// TIA Portal V16 export
// export: Created 2021-11-12T13:32:01.6049772Z, ExportSetting WithDefaults, DisplayName Totally Integrated Automation Portal, DisplayVersion V16 Update 3, DisplayName TIA Portal Version Control Interface, DisplayVersion V16 Update 2, DisplayName TIA Portal Openness, DisplayVersion V16 Update 3, DisplayName SINAMICS Startdrive Advanced, DisplayVersion V16 Update 5, DisplayName SINAMICS Startdrive G130, G150, S120, S150, SINAMICS MV, S210, DisplayVersion V16 Update 5, DisplayName SINAMICS Startdrive G110M, G120, G120C, G120D, G120P, G115D, DisplayVersion V16 Update 5, DisplayName STEP 7 Professional, DisplayVersion V16 Update 3, DisplayName STEP 7 Safety, DisplayVersion V16, DisplayName WinCC UA Professional, DisplayVersion V16 Update 3
FUNCTION_BLOCK "Station 110"   // FB53, LAD
{ S7_Optimized_Access := 'TRUE' }
VERSION : 0.1
// stored: AutoNumber true, IsIECCheckEnabled false, IsRetainMemResEnabled false, MemoryReserve 100, SetENOAutomatically false, UDAEnableTagReadback false
   VAR
      SF_Alarm1 : "STD_DI_Mon";
      SF_Alarm2 { S7_SetPoint := 'True'} : "STD_DI_Mon";
      SF_Alarm3 { S7_SetPoint := 'True'} : "STD_DI_Mon";
      SF_Alarm4 { S7_SetPoint := 'True'} : "STD_DI_Mon";
      SF_Alarm5 { S7_SetPoint := 'True'} : "STD_DI_Mon";
      SF_Alarm6 { S7_SetPoint := 'True'} : "STD_DI_Mon";
      SF_Alarm7 { S7_SetPoint := 'True'} : "STD_DI_Mon";
      SF_Alarm8 { S7_SetPoint := 'True'} : "STD_DI_Mon";
      SF_Alarm9 { S7_SetPoint := 'True'} : "STD_DI_Mon";
      SF_Alarm10 { S7_SetPoint := 'True'} : "STD_DI_Mon";
      SF_Alarm11 { S7_SetPoint := 'True'} : "STD_DI_Mon";
      SF_Alarm12 { S7_SetPoint := 'True'} : "STD_DI_Mon";
      SF_Alarm13 { S7_SetPoint := 'True'} : "STD_DI_Mon";
      SF_Alarm14 { S7_SetPoint := 'True'} : "STD_DI_Mon";
      SF_Alarm15 { S7_SetPoint := 'True'} : "STD_DI_Mon";
      SF_Alarm16 { S7_SetPoint := 'True'} : "STD_DI_Mon";
      SF_Alarm17 { S7_SetPoint := 'True'} : "STD_DI_Mon";
      SF_Alarm18 { S7_SetPoint := 'True'} : "STD_DI_Mon";
      SF_Alarm19 { S7_SetPoint := 'True'} : "STD_DI_Mon";
      SF_Alarm20 { S7_SetPoint := 'True'} : "STD_DI_Mon";
      SF_Alarm21 { S7_SetPoint := 'True'} : "STD_DI_Mon";
      SF_GL01MA02 { S7_SetPoint := 'True'} : "STD_Drive1";
      SF_UH31TA01 { S7_SetPoint := 'True'} : "STD_SERVO_FESTO_CMMT";   // Aligner - frequency convertor
      SF_UC12TA01 { S7_SetPoint := 'True'} : "STD_Siemens_G120_CU240E_2_PN";
      SF_GL01BG05 { S7_SetPoint := 'True'} : "STD_Siemens_MC_Encoder";
      SF_GL01MM01 { S7_SetPoint := 'True'} : "STD_Valve2WB";
      SF_GM01MM01 { S7_SetPoint := 'True'} : "STD_Valve2WB";
      SF_GM01MM02 { S7_SetPoint := 'True'} : "STD_Valve2WB";
      SF_GM01MM03 { S7_SetPoint := 'True'} : "STD_Valve2WB";
      SF_GM01MM04 { S7_SetPoint := 'True'} : "STD_Valve2WB";
      SS_Edge : Array[0..9] of Bool;
      SF_TON_MeasDelay { S7_SetPoint := 'True'} : TON_TIME;
      SR_ConvActPos : Real;   // Conveyor - Absolute position [mm]
   END_VAR
   VAR RETAIN
      SR_ConvStopPos : Real;   // Conveyor - Demanded position [mm]
      SB1ConvInPos { ExternalAccessible := 'False'; ExternalVisible := 'False'; ExternalWritable := 'False'} : Bool := true;   // Conveyor reached position
      SB1ConvStep : Bool;   // Step is active
      SI_SeqStepNr : UInt;   // Number of active step
      SR_UH31TA01SetPos { ExternalAccessible := 'False'; ExternalVisible := 'False'; ExternalWritable := 'False'} : Real := 550.0;   // Setpoint position [mm]
   END_VAR
   VAR
      SR_MeasuredPartLenght : Real;   // Lenght of measured part [mm]
      SI_PartType : Int;   // Part type of material
      SDIPartID : DInt;   // Part Id of material
   END_VAR
   VAR_TEMP
      TS_GL01MM01 : "UDT_DriveControl";   // Stopper - valve
      TS_GL01MA01 : "UDT_DriveControl";   // Aligner - drive
      TS_GL01MA02 : "UDT_DriveControl";   // Conveyor - drive
      TS_GM01MM01 : "UDT_DriveControl";   // Lift 1 - valve
      TS_GM01MM02 : "UDT_DriveControl";   // Lift 2 - valve
      TS_GM01MM03 : "UDT_DriveControl";   // Lift 3 - valve
      TS_GM01MM04 : "UDT_DriveControl";   // Lift 4 - valve
      TS_UC12TA01 : Struct   // Conveyor
         ReqDir1 : Bool;   // Move in direction 1
         ReqDir2 : Bool;   // Move in direction 2
         AckErr : Bool;   // Acknowledge error
         SpeedSP : Real;   // Speed setpoint
      END_STRUCT;
      TS_UH31TA01 : Struct   // Aligner
         SPPos : Int;   // Aligner - setpoint
         Mode : Int;   // Aligner - mode
         HomePos : Bool;   // Aligner - home position
         WorkPos : Bool;   // Aligner - work position
      END_STRUCT;
      TR_ConvSlowPos : Real;   // Slowing position [mm]
      "TR_ConvStepTol+" : Real;   // Upper tolerance for conveyor step [mm]
      "TR_ConvStepTol-" : Real;   // Lower tolerance for conveyor step [mm]
      "TR_UH31TA01HomeTol+" : Real;   // Upper tolerance for home position [mm]
      "TR_UH31TA01HomeTol-" : Real;   // Lower tolerance for home position [mm]
      "TR_UH31TA01WorkTol+" : Real;   // Upper tolerance for work position [mm]
      "TR_UH31TA01WorkTol-" : Real;   // Lower tolerance for work position [mm]
      TR_UH31TA01ActualPos : Real;   // Absolute position [mm]
      TR_UH31TA01HomePos : Real;   // Home position [mm]
      TR_UH31TA01WorkPos : Real;   // Working position [mm]
      TR_UH31TA01SetPos : Real;   // Setpoint position [um]
      TB1PwrOk : Bool;
      TB1EnableWork : Bool;
      TB1ResetEncoder : Bool;
   END_VAR
   VAR CONSTANT
      CI_FirstPos : Int := 28;   // Number of positions in conveyor map
      CI_MeasPos : Int := 27;   // Measuring position
      CR_ConvStepLenght : Real := 80.0;   // value [mm]
      CR_ConvSlowDist : Real := 20.0;   // Slow down - distance to stop position [mm]
      CR_ConvStepTol : Real := 2.5;   // value [mm]
      CR_EncUnitPerPulse : Real := 0.08788;   // Encoder - units per pulse [mm]
      CR_ResetEncoderPos : Real := 6080000.0;   // Position for encoder value reset [mm]
      CR_UH31TA01AligningOffset : Real := 20.0;   // value [mm]
      CR_UH31TA01HomePos : Real := 600.0;   // Home position [mm]
      CR_UH31TA01PosTol : Real := 2.0;   // Position tolerance [mm]
      CI_UH31TA01ModeRelPos : Int := 1;   // Aligner mode - relative positioning
      CI_UH31TA01ModeAbsPos : Int := 2;   // Aligner mode - absolute positioning
      CI_UH31TA01ModeGoToRefPos : Int := 4;   // Aligner mode - go to reference point
      CI_UH31TA01ModeSetRefPos : Int := 5;   // Aligner mode - set reference point
      CI_UH31TA01ModeJog : Int := 7;   // Aligner mode - jogging
      CI_SeqHomePos : UInt := 0;
      CI_SeqHomeWork : UInt := 1;
      CI_SeqWorkPos : UInt := 2;
      CI_SeqAligning : UInt := 3;
      CI_SeqMeas : UInt := 4;
      CI_SeqReturn : UInt := 5;
      CI_SeqGoHome : UInt := 6;
      CI_MeasOffset : Real := 55.5;
   END_VAR
   // // SF_UH31TA01.SF_SINA_POS : Copyright (C) Siemens AG 2012. All Rights Reserved. Confidential-------------------------------------------------------------------------------------- SINA_POS: Positionierung mit dem Antriebsbaustein SINAMICS S110/G120 <-> S7-1100------------------------------------------------------------------------------------- Ersteller: Siemens AG Erlangen A&D MC PM Datum: 07.07.10 Vers.:2.1Änderung: J.B. Typical Team 18.12.12 2.2 Umsetzung in SCL / TIA Änderung: J.B. Typical Team 18.04.13 2.3 Bei Betriebsart "Referenzieren - Referenzpunkt setzen" nicht intern setzen sondern Eingang #Execute abfragen als StartbedingungÄnderung: J.B. Typical Team 29.04.13 2.4 1. Off1 möglich bei ungültige Betriebsart 2. Referenzpunkt setzen Exceute übernehmen 3. Fehlermeldung ausgeben bei Wechel ohne Beendigung der Betriebsart 4. "Q" an den Ausgänge entfernen 5. Neuer Ausgang PwrInhibit Änderung: J.B. Typical Team 14.05.13 2.5 Fehlerbehebung und Defaultwerte ändernÄnderung: J.B. Typical Team 28.06.13 2.6 HW-Zugriffsermittlung über LOG2MODÄnderung: J.B. Typical Team 18.07.13 2.7 HW-Zugriffsermittlung über zwei HW-EingängeÄnderung: J.B. Typical Team 18.09.13 2.8 Konvertierungsfehler behobenÄnderung: J.B. Typical Team 25.09.13 2.9 Bei Betriebswechsel von 3 nach 6 darf MidStart nicht sitzenÄnderung: J.B. Typical Team 31.03.14 3.0 In der Betriebsart 1-3 und 6 darf MidTrTyp nicht sitzenÄnderung: J.B. Typical Team 25.06.14 3.1 Das Quittierbit "AckFlt" immer durchreichenÄnderung: J.B. Typical Team 30.07.14 4.0 Festlegung auf einheitlicher neuer Version 4.0Änderung: J.B. Typical Team 07.11.14 4.1 Fehlerbehebung falsche Zuweisung von Off1 bei Mode 4 und Mode 8(DriveLib V4 - RQ 346046)Änderung: F.G. Typical Team 16.04.15 4.2 Anzahl der Zyklen die auf die Rückmeldung fliegendes Ref. gewartet wird verdoppelt (siRetryMax = 10) (DriveLib V4 - RQ 367986)Änderung: F.G. Typical Team 15.09.15 4.3 Anzahl der Zyklen die auf die Rückmeldung fliegendes Ref. gewartet noch einmal um 5 erhöht (siRetryMax = 15) (DriveLib V4 - RQ 367986)Änderung: F.G. Typical Team 15.09.15 4.4 Abfrage des richtigen Bits im EPosZSW1 (Zeile 1394)es muss das Bit12 und nicht das Bit 11 abgefragt werden (DriveLib V4 - RQ 367986)Änderung: F.G. Typical Team 03.12.15 4.5 1. Ein-/Ausgänge an Programmierleitfaden für TIA-Portal angepasst Zusätzlicher Eingang um alle Bits in den STWs zu bedienen 2. Warnung durch Initialisierung elimininiertÄnderung: F.G. Typical Team 13.09.16 4.6 Ausgabewerte am Ausgang "Status" angepasst Änderung: G.F. Typical Team 11.01.17 5.0 - Festlegung auf einheitlicher neuer Version 5.0 Bibliothek V7Funktion: Positionierung mit dem Antriebsbaustein SINAMICS S110/G120 <-> S7-1100********************************************************************************************************************************************************************************************************************************FB283***********************************************************************************************************************************************************************************************************************************
   VAR_TEMP   // added for the SCL form of the ladder/FBD networks
      _w1 : Bool;
      _w2 : Bool;
      _w3 : Bool;
      _w4 : Bool;
      _w5 : Bool;
      _w6 : Bool;
      _w7 : Bool;
      _w8 : Bool;
      _w9 : Bool;
      _w10 : Bool;
      _w11 : Bool;
      _w12 : Bool;
      _w13 : Bool;
      _w14 : Bool;
      _w15 : Bool;
      _w16 : Bool;
      _w17 : Bool;
      _w18 : Bool;
      _w19 : Bool;
      _w20 : Bool;
      _w21 : Bool;
      _w22 : Bool;
      _w23 : Bool;
      _w24 : Bool;
      _w25 : Bool;
      _w26 : Bool;
      _w27 : Bool;
      _w28 : Bool;
      _w29 : Bool;
   END_VAR
BEGIN

REGION Network 1: Reset temporary variables
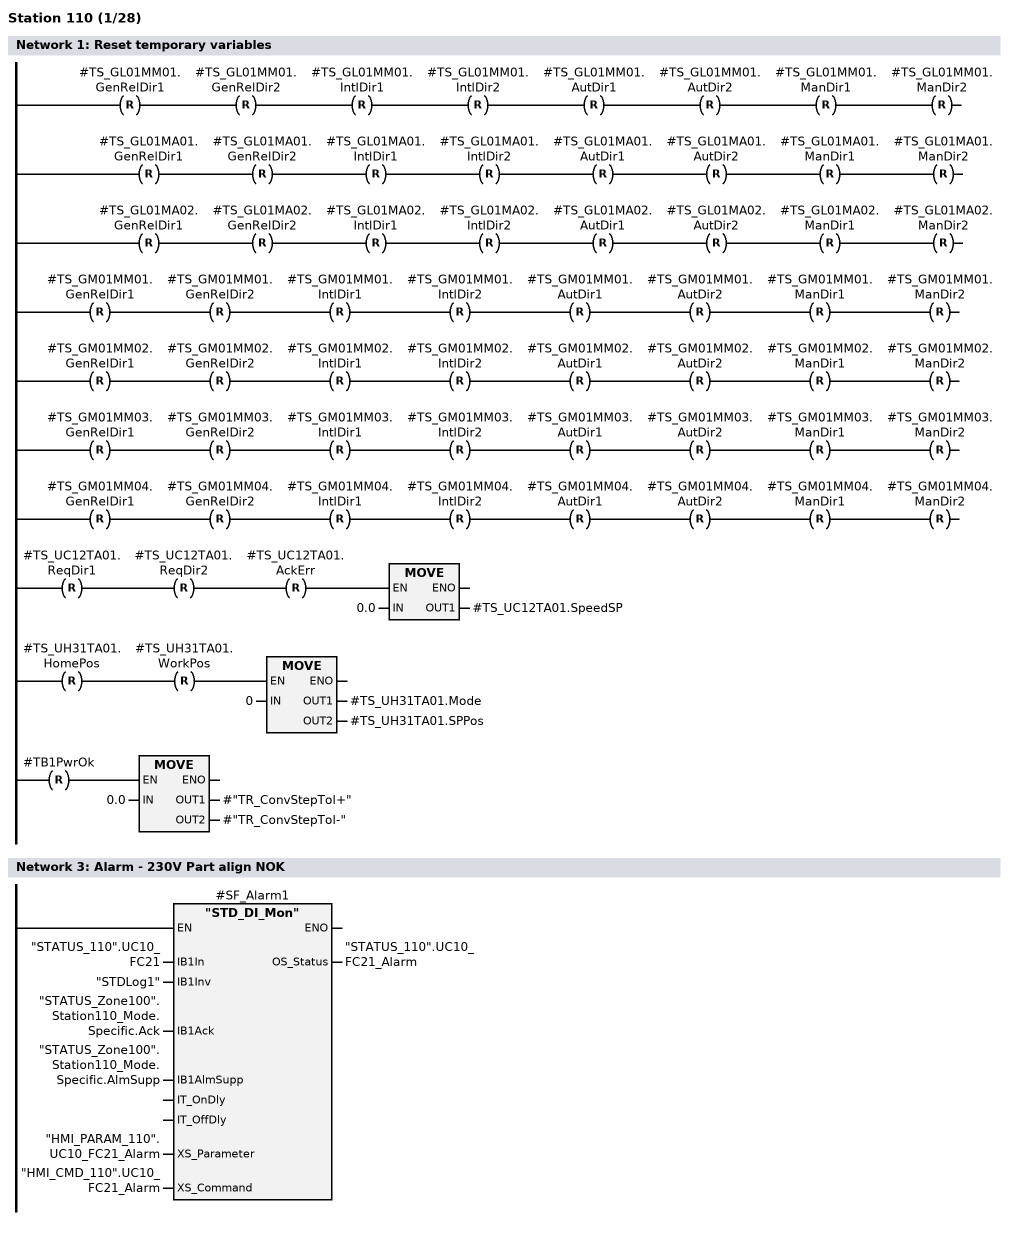
   RUNG wire#powerrail
      R_Coil( #TS_GL01MM01.GenRelDir1 )
      R_Coil( #TS_GL01MM01.GenRelDir2 )
      R_Coil( #TS_GL01MM01.IntlDir1 )
      R_Coil( #TS_GL01MM01.IntlDir2 )
      R_Coil( #TS_GL01MM01.AutDir1 )
      R_Coil( #TS_GL01MM01.AutDir2 )
      R_Coil( #TS_GL01MM01.ManDir1 )
      R_Coil( #TS_GL01MM01.ManDir2 )
   END_RUNG
   RUNG wire#powerrail
      R_Coil( #TS_GL01MA01.GenRelDir1 )
      R_Coil( #TS_GL01MA01.GenRelDir2 )
      R_Coil( #TS_GL01MA01.IntlDir1 )
      R_Coil( #TS_GL01MA01.IntlDir2 )
      R_Coil( #TS_GL01MA01.AutDir1 )
      R_Coil( #TS_GL01MA01.AutDir2 )
      R_Coil( #TS_GL01MA01.ManDir1 )
      R_Coil( #TS_GL01MA01.ManDir2 )
   END_RUNG
   RUNG wire#powerrail
      R_Coil( #TS_GL01MA02.GenRelDir1 )
      R_Coil( #TS_GL01MA02.GenRelDir2 )
      R_Coil( #TS_GL01MA02.IntlDir1 )
      R_Coil( #TS_GL01MA02.IntlDir2 )
      R_Coil( #TS_GL01MA02.AutDir1 )
      R_Coil( #TS_GL01MA02.AutDir2 )
      R_Coil( #TS_GL01MA02.ManDir1 )
      R_Coil( #TS_GL01MA02.ManDir2 )
   END_RUNG
   RUNG wire#powerrail
      R_Coil( #TS_GM01MM01.GenRelDir1 )
      R_Coil( #TS_GM01MM01.GenRelDir2 )
      R_Coil( #TS_GM01MM01.IntlDir1 )
      R_Coil( #TS_GM01MM01.IntlDir2 )
      R_Coil( #TS_GM01MM01.AutDir1 )
      R_Coil( #TS_GM01MM01.AutDir2 )
      R_Coil( #TS_GM01MM01.ManDir1 )
      R_Coil( #TS_GM01MM01.ManDir2 )
   END_RUNG
   RUNG wire#powerrail
      R_Coil( #TS_GM01MM02.GenRelDir1 )
      R_Coil( #TS_GM01MM02.GenRelDir2 )
      R_Coil( #TS_GM01MM02.IntlDir1 )
      R_Coil( #TS_GM01MM02.IntlDir2 )
      R_Coil( #TS_GM01MM02.AutDir1 )
      R_Coil( #TS_GM01MM02.AutDir2 )
      R_Coil( #TS_GM01MM02.ManDir1 )
      R_Coil( #TS_GM01MM02.ManDir2 )
   END_RUNG
   RUNG wire#powerrail
      R_Coil( #TS_GM01MM03.GenRelDir1 )
      R_Coil( #TS_GM01MM03.GenRelDir2 )
      R_Coil( #TS_GM01MM03.IntlDir1 )
      R_Coil( #TS_GM01MM03.IntlDir2 )
      R_Coil( #TS_GM01MM03.AutDir1 )
      R_Coil( #TS_GM01MM03.AutDir2 )
      R_Coil( #TS_GM01MM03.ManDir1 )
      R_Coil( #TS_GM01MM03.ManDir2 )
   END_RUNG
   RUNG wire#powerrail
      R_Coil( #TS_GM01MM04.GenRelDir1 )
      R_Coil( #TS_GM01MM04.GenRelDir2 )
      R_Coil( #TS_GM01MM04.IntlDir1 )
      R_Coil( #TS_GM01MM04.IntlDir2 )
      R_Coil( #TS_GM01MM04.AutDir1 )
      R_Coil( #TS_GM01MM04.AutDir2 )
      R_Coil( #TS_GM01MM04.ManDir1 )
      R_Coil( #TS_GM01MM04.ManDir2 )
   END_RUNG
   RUNG wire#powerrail
      R_Coil( #TS_UC12TA01.ReqDir1 )
      R_Coil( #TS_UC12TA01.ReqDir2 )
      R_Coil( #TS_UC12TA01.AckErr )
      Move(in := 0.0, out1 => #TS_UC12TA01.SpeedSP)
   END_RUNG
   RUNG wire#powerrail
      R_Coil( #TS_UH31TA01.HomePos )
      R_Coil( #TS_UH31TA01.WorkPos )
      Move(in := 0, out1 => #TS_UH31TA01.Mode, out2 => #TS_UH31TA01.SPPos)
   END_RUNG
   RUNG wire#powerrail
      R_Coil( #TB1PwrOk )
      Move(in := 0.0, out1 => #"TR_ConvStepTol+", out2 => #"TR_ConvStepTol-")
   END_RUNG
   // the same network as SCL:
   #TS_GL01MM01.GenRelDir1 := FALSE;
   #TS_GL01MM01.GenRelDir2 := FALSE;
   #TS_GL01MM01.IntlDir1 := FALSE;
   #TS_GL01MM01.IntlDir2 := FALSE;
   #TS_GL01MM01.AutDir1 := FALSE;
   #TS_GL01MM01.AutDir2 := FALSE;
   #TS_GL01MM01.ManDir1 := FALSE;
   #TS_GL01MM01.ManDir2 := FALSE;
   #TS_GL01MA01.GenRelDir1 := FALSE;
   #TS_GL01MA01.GenRelDir2 := FALSE;
   #TS_GL01MA01.IntlDir1 := FALSE;
   #TS_GL01MA01.IntlDir2 := FALSE;
   #TS_GL01MA01.AutDir1 := FALSE;
   #TS_GL01MA01.AutDir2 := FALSE;
   #TS_GL01MA01.ManDir1 := FALSE;
   #TS_GL01MA01.ManDir2 := FALSE;
   #TS_GL01MA02.GenRelDir1 := FALSE;
   #TS_GL01MA02.GenRelDir2 := FALSE;
   #TS_GL01MA02.IntlDir1 := FALSE;
   #TS_GL01MA02.IntlDir2 := FALSE;
   #TS_GL01MA02.AutDir1 := FALSE;
   #TS_GL01MA02.AutDir2 := FALSE;
   #TS_GL01MA02.ManDir1 := FALSE;
   #TS_GL01MA02.ManDir2 := FALSE;
   #TS_GM01MM01.GenRelDir1 := FALSE;
   #TS_GM01MM01.GenRelDir2 := FALSE;
   #TS_GM01MM01.IntlDir1 := FALSE;
   #TS_GM01MM01.IntlDir2 := FALSE;
   #TS_GM01MM01.AutDir1 := FALSE;
   #TS_GM01MM01.AutDir2 := FALSE;
   #TS_GM01MM01.ManDir1 := FALSE;
   #TS_GM01MM01.ManDir2 := FALSE;
   #TS_GM01MM02.GenRelDir1 := FALSE;
   #TS_GM01MM02.GenRelDir2 := FALSE;
   #TS_GM01MM02.IntlDir1 := FALSE;
   #TS_GM01MM02.IntlDir2 := FALSE;
   #TS_GM01MM02.AutDir1 := FALSE;
   #TS_GM01MM02.AutDir2 := FALSE;
   #TS_GM01MM02.ManDir1 := FALSE;
   #TS_GM01MM02.ManDir2 := FALSE;
   #TS_GM01MM03.GenRelDir1 := FALSE;
   #TS_GM01MM03.GenRelDir2 := FALSE;
   #TS_GM01MM03.IntlDir1 := FALSE;
   #TS_GM01MM03.IntlDir2 := FALSE;
   #TS_GM01MM03.AutDir1 := FALSE;
   #TS_GM01MM03.AutDir2 := FALSE;
   #TS_GM01MM03.ManDir1 := FALSE;
   #TS_GM01MM03.ManDir2 := FALSE;
   #TS_GM01MM04.GenRelDir1 := FALSE;
   #TS_GM01MM04.GenRelDir2 := FALSE;
   #TS_GM01MM04.IntlDir1 := FALSE;
   #TS_GM01MM04.IntlDir2 := FALSE;
   #TS_GM01MM04.AutDir1 := FALSE;
   #TS_GM01MM04.AutDir2 := FALSE;
   #TS_GM01MM04.ManDir1 := FALSE;
   #TS_GM01MM04.ManDir2 := FALSE;
   #TS_UC12TA01.ReqDir1 := FALSE;
   #TS_UC12TA01.ReqDir2 := FALSE;
   #TS_UC12TA01.AckErr := FALSE;
   #TS_UC12TA01.SpeedSP := 0.0;
   #TS_UH31TA01.HomePos := FALSE;
   #TS_UH31TA01.WorkPos := FALSE;
   #TS_UH31TA01.Mode := 0;
   #TS_UH31TA01.SPPos := 0;
   #TB1PwrOk := FALSE;
   #"TR_ConvStepTol+" := 0.0;
   #"TR_ConvStepTol-" := 0.0;
END_REGION

REGION Network 2: *************** Alarms ***************
END_REGION

REGION Network 3: Alarm - 230V Part align NOK
   RUNG wire#powerrail
      #SF_Alarm1(IB1In := "STATUS_110".UC10_FC21, IB1Inv := "STDLog1", IB1Ack := "STATUS_Zone100".Station110_Mode.Specific.Ack, IB1AlmSupp := "STATUS_Zone100".Station110_Mode.Specific.AlmSupp, IT_OnDly :=, IT_OffDly :=, XS_Parameter := "HMI_PARAM_110".UC10_FC21_Alarm, XS_Command := "HMI_CMD_110".UC10_FC21_Alarm, OS_Status => "STATUS_110".UC10_FC21_Alarm)
   END_RUNG
   // the same network as SCL:
   #SF_Alarm1(IB1In := "STATUS_110".UC10_FC21,   // "STD_DI_Mon"
              IB1Inv := "STDLog1",
              IB1Ack := "STATUS_Zone100".Station110_Mode.Specific.Ack,
              IB1AlmSupp := "STATUS_Zone100".Station110_Mode.Specific.AlmSupp,
              XS_Parameter := "HMI_PARAM_110".UC10_FC21_Alarm,
              XS_Command := "HMI_CMD_110".UC10_FC21_Alarm,
              OS_Status => "STATUS_110".UC10_FC21_Alarm);
END_REGION

REGION Network 4: Alarm - 400V Conveyor NOK
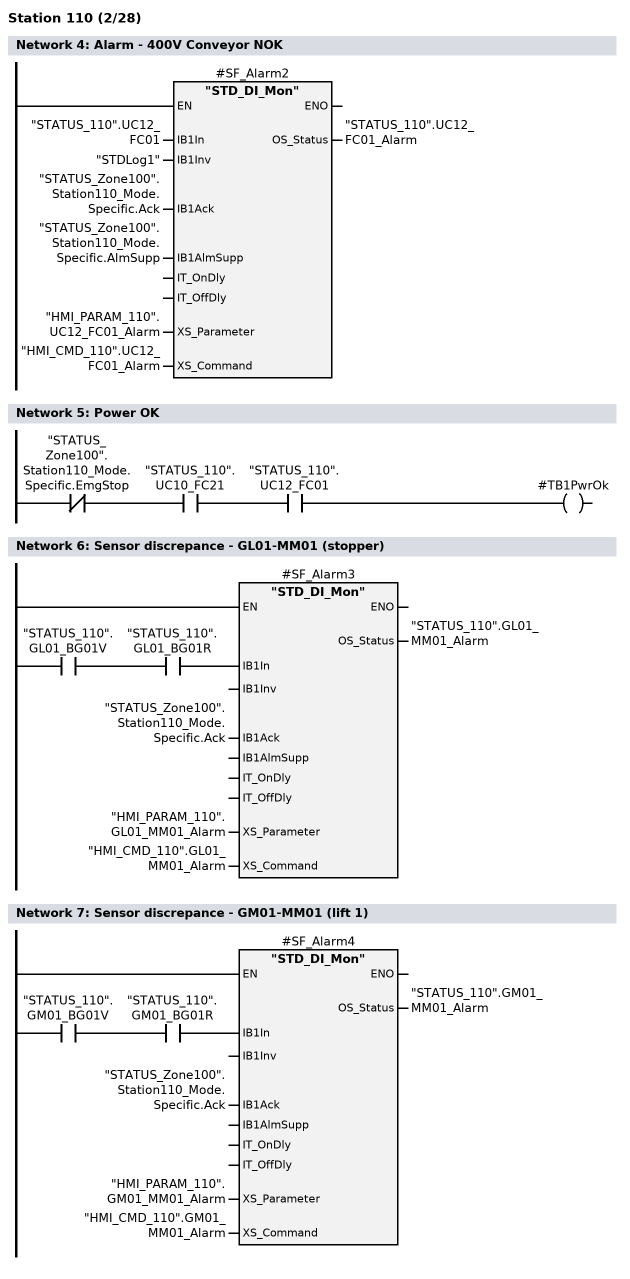
   RUNG wire#powerrail
      #SF_Alarm2(IB1In := "STATUS_110".UC12_FC01, IB1Inv := "STDLog1", IB1Ack := "STATUS_Zone100".Station110_Mode.Specific.Ack, IB1AlmSupp := "STATUS_Zone100".Station110_Mode.Specific.AlmSupp, IT_OnDly :=, IT_OffDly :=, XS_Parameter := "HMI_PARAM_110".UC12_FC01_Alarm, XS_Command := "HMI_CMD_110".UC12_FC01_Alarm, OS_Status => "STATUS_110".UC12_FC01_Alarm)
   END_RUNG
   // the same network as SCL:
   #SF_Alarm2(IB1In := "STATUS_110".UC12_FC01,   // "STD_DI_Mon"
              IB1Inv := "STDLog1",
              IB1Ack := "STATUS_Zone100".Station110_Mode.Specific.Ack,
              IB1AlmSupp := "STATUS_Zone100".Station110_Mode.Specific.AlmSupp,
              XS_Parameter := "HMI_PARAM_110".UC12_FC01_Alarm,
              XS_Command := "HMI_CMD_110".UC12_FC01_Alarm,
              OS_Status => "STATUS_110".UC12_FC01_Alarm);
END_REGION

REGION Network 5: Power OK
   RUNG wire#powerrail
      I_Contact( "STATUS_Zone100".Station110_Mode.Specific.EmgStop )
      Contact( "STATUS_110".UC10_FC21 )
      Contact( "STATUS_110".UC12_FC01 )
      Coil( #TB1PwrOk )
   END_RUNG
   // the same network as SCL:
   #TB1PwrOk := NOT "STATUS_Zone100".Station110_Mode.Specific.EmgStop AND "STATUS_110".UC10_FC21 AND "STATUS_110".UC12_FC01;
END_REGION

REGION Network 6: Sensor discrepance - GL01-MM01 (stopper)
   RUNG wire#powerrail
      #SF_Alarm3(IB1In := wire#w1, IB1Inv :=, IB1Ack := "STATUS_Zone100".Station110_Mode.Specific.Ack, IB1AlmSupp :=, IT_OnDly :=, IT_OffDly :=, XS_Parameter := "HMI_PARAM_110".GL01_MM01_Alarm, XS_Command := "HMI_CMD_110".GL01_MM01_Alarm, OS_Status => "STATUS_110".GL01_MM01_Alarm)
   END_RUNG
   RUNG wire#powerrail
      Contact( "STATUS_110".GL01_BG01V )
      Contact( "STATUS_110".GL01_BG01R )
   END_RUNG wire#w1
   // the same network as SCL:
   #SF_Alarm3(IB1In := "STATUS_110".GL01_BG01V AND "STATUS_110".GL01_BG01R,   // "STD_DI_Mon"
              IB1Ack := "STATUS_Zone100".Station110_Mode.Specific.Ack,
              XS_Parameter := "HMI_PARAM_110".GL01_MM01_Alarm,
              XS_Command := "HMI_CMD_110".GL01_MM01_Alarm,
              OS_Status => "STATUS_110".GL01_MM01_Alarm);
END_REGION

REGION Network 7: Sensor discrepance - GM01-MM01 (lift 1)
   RUNG wire#powerrail
      #SF_Alarm4(IB1In := wire#w1, IB1Inv :=, IB1Ack := "STATUS_Zone100".Station110_Mode.Specific.Ack, IB1AlmSupp :=, IT_OnDly :=, IT_OffDly :=, XS_Parameter := "HMI_PARAM_110".GM01_MM01_Alarm, XS_Command := "HMI_CMD_110".GM01_MM01_Alarm, OS_Status => "STATUS_110".GM01_MM01_Alarm)
   END_RUNG
   RUNG wire#powerrail
      Contact( "STATUS_110".GM01_BG01V )
      Contact( "STATUS_110".GM01_BG01R )
   END_RUNG wire#w1
   // the same network as SCL:
   #SF_Alarm4(IB1In := "STATUS_110".GM01_BG01V AND "STATUS_110".GM01_BG01R,   // "STD_DI_Mon"
              IB1Ack := "STATUS_Zone100".Station110_Mode.Specific.Ack,
              XS_Parameter := "HMI_PARAM_110".GM01_MM01_Alarm,
              XS_Command := "HMI_CMD_110".GM01_MM01_Alarm,
              OS_Status => "STATUS_110".GM01_MM01_Alarm);
END_REGION

REGION Network 8: Sensor discrepance - GM01-MM02 (lift 2)
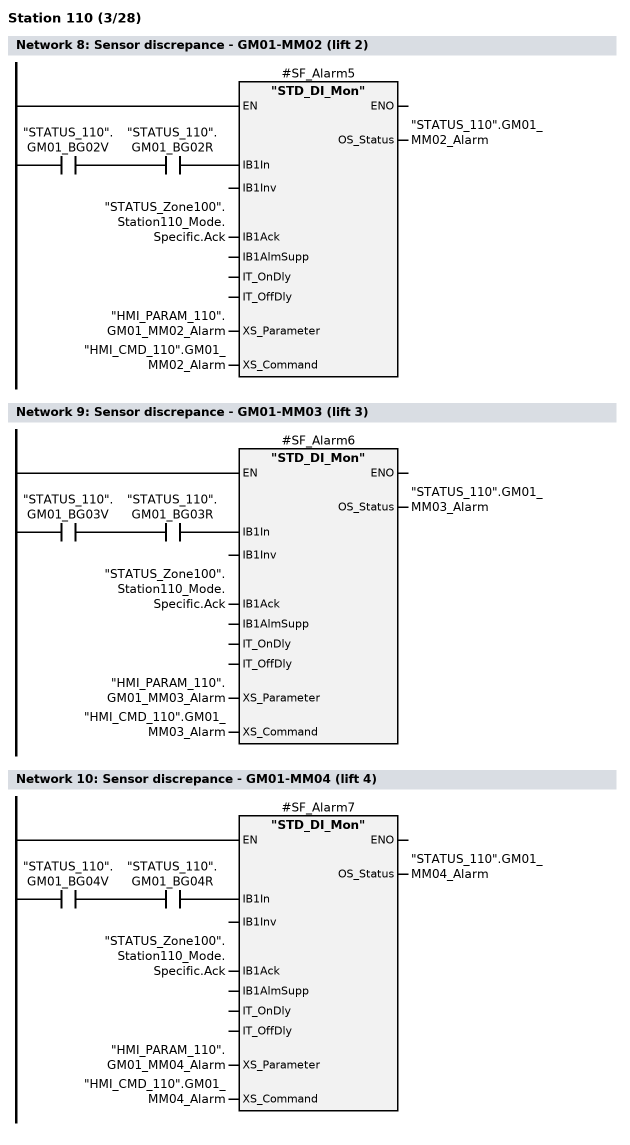
   RUNG wire#powerrail
      #SF_Alarm5(IB1In := wire#w1, IB1Inv :=, IB1Ack := "STATUS_Zone100".Station110_Mode.Specific.Ack, IB1AlmSupp :=, IT_OnDly :=, IT_OffDly :=, XS_Parameter := "HMI_PARAM_110".GM01_MM02_Alarm, XS_Command := "HMI_CMD_110".GM01_MM02_Alarm, OS_Status => "STATUS_110".GM01_MM02_Alarm)
   END_RUNG
   RUNG wire#powerrail
      Contact( "STATUS_110".GM01_BG02V )
      Contact( "STATUS_110".GM01_BG02R )
   END_RUNG wire#w1
   // the same network as SCL:
   #SF_Alarm5(IB1In := "STATUS_110".GM01_BG02V AND "STATUS_110".GM01_BG02R,   // "STD_DI_Mon"
              IB1Ack := "STATUS_Zone100".Station110_Mode.Specific.Ack,
              XS_Parameter := "HMI_PARAM_110".GM01_MM02_Alarm,
              XS_Command := "HMI_CMD_110".GM01_MM02_Alarm,
              OS_Status => "STATUS_110".GM01_MM02_Alarm);
END_REGION

REGION Network 9: Sensor discrepance - GM01-MM03 (lift 3)
   RUNG wire#powerrail
      #SF_Alarm6(IB1In := wire#w1, IB1Inv :=, IB1Ack := "STATUS_Zone100".Station110_Mode.Specific.Ack, IB1AlmSupp :=, IT_OnDly :=, IT_OffDly :=, XS_Parameter := "HMI_PARAM_110".GM01_MM03_Alarm, XS_Command := "HMI_CMD_110".GM01_MM03_Alarm, OS_Status => "STATUS_110".GM01_MM03_Alarm)
   END_RUNG
   RUNG wire#powerrail
      Contact( "STATUS_110".GM01_BG03V )
      Contact( "STATUS_110".GM01_BG03R )
   END_RUNG wire#w1
   // the same network as SCL:
   #SF_Alarm6(IB1In := "STATUS_110".GM01_BG03V AND "STATUS_110".GM01_BG03R,   // "STD_DI_Mon"
              IB1Ack := "STATUS_Zone100".Station110_Mode.Specific.Ack,
              XS_Parameter := "HMI_PARAM_110".GM01_MM03_Alarm,
              XS_Command := "HMI_CMD_110".GM01_MM03_Alarm,
              OS_Status => "STATUS_110".GM01_MM03_Alarm);
END_REGION

REGION Network 10: Sensor discrepance - GM01-MM04 (lift 4)
   RUNG wire#powerrail
      #SF_Alarm7(IB1In := wire#w1, IB1Inv :=, IB1Ack := "STATUS_Zone100".Station110_Mode.Specific.Ack, IB1AlmSupp :=, IT_OnDly :=, IT_OffDly :=, XS_Parameter := "HMI_PARAM_110".GM01_MM04_Alarm, XS_Command := "HMI_CMD_110".GM01_MM04_Alarm, OS_Status => "STATUS_110".GM01_MM04_Alarm)
   END_RUNG
   RUNG wire#powerrail
      Contact( "STATUS_110".GM01_BG04V )
      Contact( "STATUS_110".GM01_BG04R )
   END_RUNG wire#w1
   // the same network as SCL:
   #SF_Alarm7(IB1In := "STATUS_110".GM01_BG04V AND "STATUS_110".GM01_BG04R,   // "STD_DI_Mon"
              IB1Ack := "STATUS_Zone100".Station110_Mode.Specific.Ack,
              XS_Parameter := "HMI_PARAM_110".GM01_MM04_Alarm,
              XS_Command := "HMI_CMD_110".GM01_MM04_Alarm,
              OS_Status => "STATUS_110".GM01_MM04_Alarm);
END_REGION

REGION Network 11: Alarm - Part in stopping position not on map
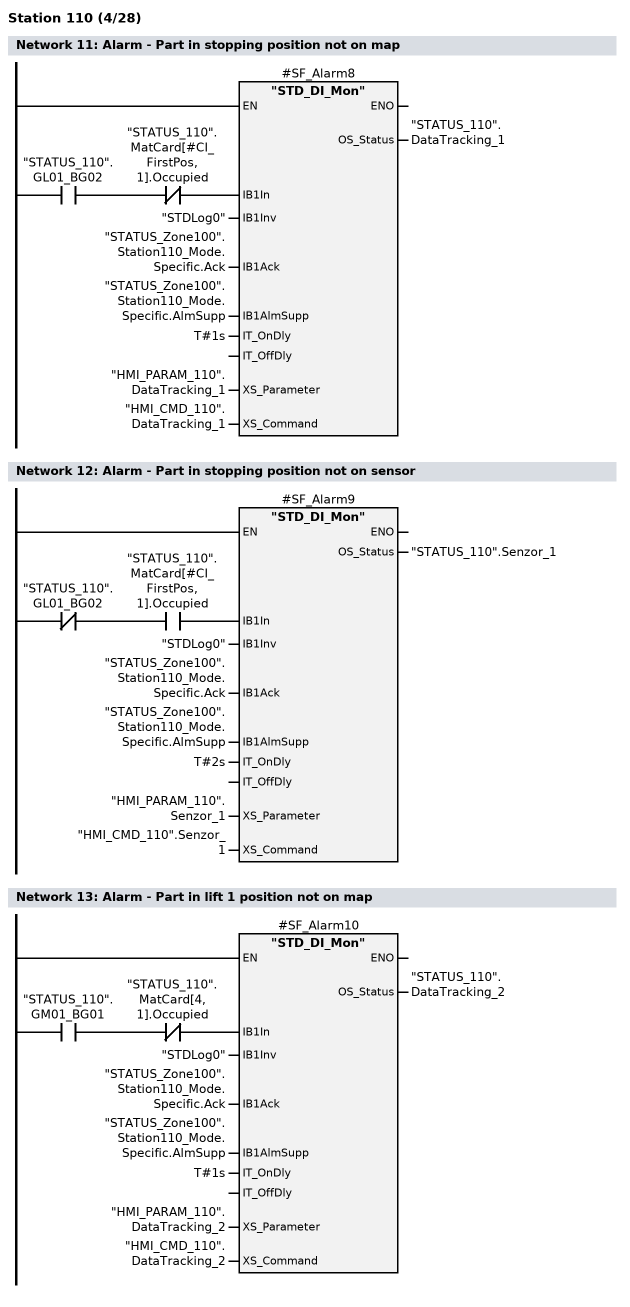
   RUNG wire#powerrail
      #SF_Alarm8(IB1In := wire#w1, IB1Inv := "STDLog0", IB1Ack := "STATUS_Zone100".Station110_Mode.Specific.Ack, IB1AlmSupp := "STATUS_Zone100".Station110_Mode.Specific.AlmSupp, IT_OnDly := T#1s, IT_OffDly :=, XS_Parameter := "HMI_PARAM_110".DataTracking_1, XS_Command := "HMI_CMD_110".DataTracking_1, OS_Status => "STATUS_110".DataTracking_1)
   END_RUNG
   RUNG wire#powerrail
      Contact( "STATUS_110".GL01_BG02 )
      I_Contact( "STATUS_110".MatCard[#CI_FirstPos, 1].Occupied )
   END_RUNG wire#w1
   // the same network as SCL:
   #SF_Alarm8(IB1In := "STATUS_110".GL01_BG02 AND NOT "STATUS_110".MatCard[#CI_FirstPos, 1].Occupied,   // "STD_DI_Mon"
              IB1Inv := "STDLog0",
              IB1Ack := "STATUS_Zone100".Station110_Mode.Specific.Ack,
              IB1AlmSupp := "STATUS_Zone100".Station110_Mode.Specific.AlmSupp,
              IT_OnDly := T#1s,
              XS_Parameter := "HMI_PARAM_110".DataTracking_1,
              XS_Command := "HMI_CMD_110".DataTracking_1,
              OS_Status => "STATUS_110".DataTracking_1);
END_REGION

REGION Network 12: Alarm - Part in stopping position not on sensor
   RUNG wire#powerrail
      #SF_Alarm9(IB1In := wire#w1, IB1Inv := "STDLog0", IB1Ack := "STATUS_Zone100".Station110_Mode.Specific.Ack, IB1AlmSupp := "STATUS_Zone100".Station110_Mode.Specific.AlmSupp, IT_OnDly := T#2s, IT_OffDly :=, XS_Parameter := "HMI_PARAM_110".Senzor_1, XS_Command := "HMI_CMD_110".Senzor_1, OS_Status => "STATUS_110".Senzor_1)
   END_RUNG
   RUNG wire#powerrail
      I_Contact( "STATUS_110".GL01_BG02 )
      Contact( "STATUS_110".MatCard[#CI_FirstPos, 1].Occupied )
   END_RUNG wire#w1
   // the same network as SCL:
   #SF_Alarm9(IB1In := NOT "STATUS_110".GL01_BG02 AND "STATUS_110".MatCard[#CI_FirstPos, 1].Occupied,   // "STD_DI_Mon"
              IB1Inv := "STDLog0",
              IB1Ack := "STATUS_Zone100".Station110_Mode.Specific.Ack,
              IB1AlmSupp := "STATUS_Zone100".Station110_Mode.Specific.AlmSupp,
              IT_OnDly := T#2s,
              XS_Parameter := "HMI_PARAM_110".Senzor_1,
              XS_Command := "HMI_CMD_110".Senzor_1,
              OS_Status => "STATUS_110".Senzor_1);
END_REGION

REGION Network 13: Alarm - Part in lift 1 position not on map
   RUNG wire#powerrail
      #SF_Alarm10(IB1In := wire#w1, IB1Inv := "STDLog0", IB1Ack := "STATUS_Zone100".Station110_Mode.Specific.Ack, IB1AlmSupp := "STATUS_Zone100".Station110_Mode.Specific.AlmSupp, IT_OnDly := T#1s, IT_OffDly :=, XS_Parameter := "HMI_PARAM_110".DataTracking_2, XS_Command := "HMI_CMD_110".DataTracking_2, OS_Status => "STATUS_110".DataTracking_2)
   END_RUNG
   RUNG wire#powerrail
      Contact( "STATUS_110".GM01_BG01 )
      I_Contact( "STATUS_110".MatCard[4, 1].Occupied )
   END_RUNG wire#w1
   // the same network as SCL:
   #SF_Alarm10(IB1In := "STATUS_110".GM01_BG01 AND NOT "STATUS_110".MatCard[4, 1].Occupied,   // "STD_DI_Mon"
               IB1Inv := "STDLog0",
               IB1Ack := "STATUS_Zone100".Station110_Mode.Specific.Ack,
               IB1AlmSupp := "STATUS_Zone100".Station110_Mode.Specific.AlmSupp,
               IT_OnDly := T#1s,
               XS_Parameter := "HMI_PARAM_110".DataTracking_2,
               XS_Command := "HMI_CMD_110".DataTracking_2,
               OS_Status => "STATUS_110".DataTracking_2);
END_REGION

REGION Network 14: Alarm - Part in lift 1 position not on sensor
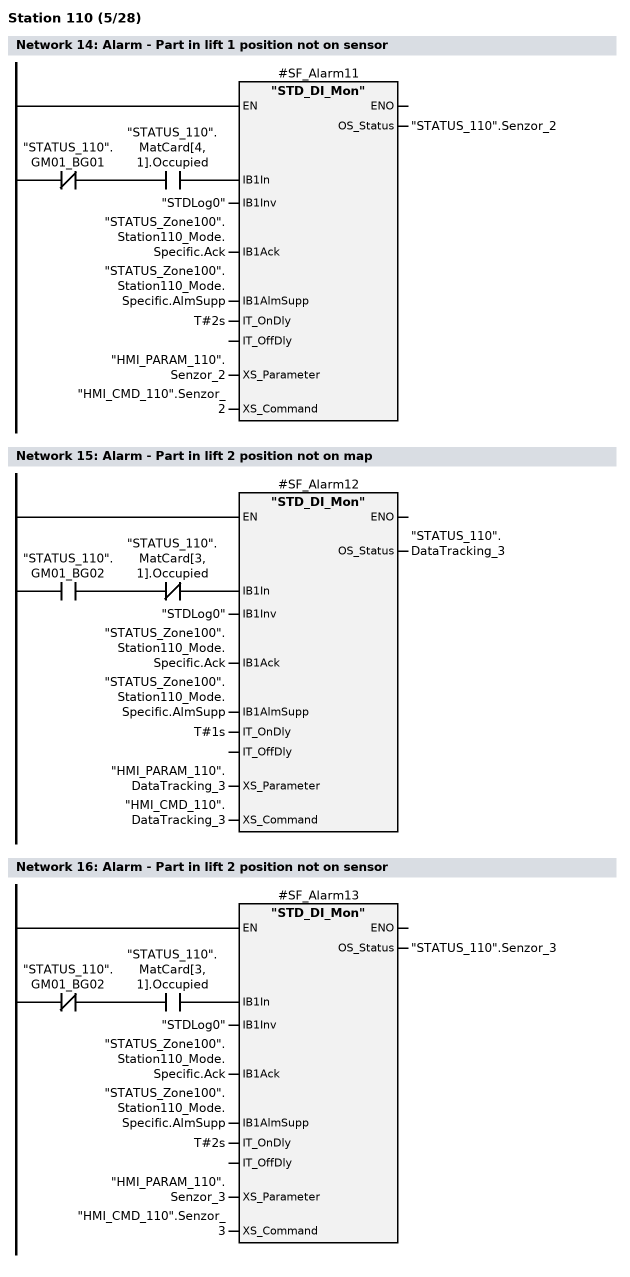
   RUNG wire#powerrail
      #SF_Alarm11(IB1In := wire#w1, IB1Inv := "STDLog0", IB1Ack := "STATUS_Zone100".Station110_Mode.Specific.Ack, IB1AlmSupp := "STATUS_Zone100".Station110_Mode.Specific.AlmSupp, IT_OnDly := T#2s, IT_OffDly :=, XS_Parameter := "HMI_PARAM_110".Senzor_2, XS_Command := "HMI_CMD_110".Senzor_2, OS_Status => "STATUS_110".Senzor_2)
   END_RUNG
   RUNG wire#powerrail
      I_Contact( "STATUS_110".GM01_BG01 )
      Contact( "STATUS_110".MatCard[4, 1].Occupied )
   END_RUNG wire#w1
   // the same network as SCL:
   #SF_Alarm11(IB1In := NOT "STATUS_110".GM01_BG01 AND "STATUS_110".MatCard[4, 1].Occupied,   // "STD_DI_Mon"
               IB1Inv := "STDLog0",
               IB1Ack := "STATUS_Zone100".Station110_Mode.Specific.Ack,
               IB1AlmSupp := "STATUS_Zone100".Station110_Mode.Specific.AlmSupp,
               IT_OnDly := T#2s,
               XS_Parameter := "HMI_PARAM_110".Senzor_2,
               XS_Command := "HMI_CMD_110".Senzor_2,
               OS_Status => "STATUS_110".Senzor_2);
END_REGION

REGION Network 15: Alarm - Part in lift 2 position not on map
   RUNG wire#powerrail
      #SF_Alarm12(IB1In := wire#w1, IB1Inv := "STDLog0", IB1Ack := "STATUS_Zone100".Station110_Mode.Specific.Ack, IB1AlmSupp := "STATUS_Zone100".Station110_Mode.Specific.AlmSupp, IT_OnDly := T#1s, IT_OffDly :=, XS_Parameter := "HMI_PARAM_110".DataTracking_3, XS_Command := "HMI_CMD_110".DataTracking_3, OS_Status => "STATUS_110".DataTracking_3)
   END_RUNG
   RUNG wire#powerrail
      Contact( "STATUS_110".GM01_BG02 )
      I_Contact( "STATUS_110".MatCard[3, 1].Occupied )
   END_RUNG wire#w1
   // the same network as SCL:
   #SF_Alarm12(IB1In := "STATUS_110".GM01_BG02 AND NOT "STATUS_110".MatCard[3, 1].Occupied,   // "STD_DI_Mon"
               IB1Inv := "STDLog0",
               IB1Ack := "STATUS_Zone100".Station110_Mode.Specific.Ack,
               IB1AlmSupp := "STATUS_Zone100".Station110_Mode.Specific.AlmSupp,
               IT_OnDly := T#1s,
               XS_Parameter := "HMI_PARAM_110".DataTracking_3,
               XS_Command := "HMI_CMD_110".DataTracking_3,
               OS_Status => "STATUS_110".DataTracking_3);
END_REGION

REGION Network 16: Alarm - Part in lift 2 position not on sensor
   RUNG wire#powerrail
      #SF_Alarm13(IB1In := wire#w1, IB1Inv := "STDLog0", IB1Ack := "STATUS_Zone100".Station110_Mode.Specific.Ack, IB1AlmSupp := "STATUS_Zone100".Station110_Mode.Specific.AlmSupp, IT_OnDly := T#2s, IT_OffDly :=, XS_Parameter := "HMI_PARAM_110".Senzor_3, XS_Command := "HMI_CMD_110".Senzor_3, OS_Status => "STATUS_110".Senzor_3)
   END_RUNG
   RUNG wire#powerrail
      I_Contact( "STATUS_110".GM01_BG02 )
      Contact( "STATUS_110".MatCard[3, 1].Occupied )
   END_RUNG wire#w1
   // the same network as SCL:
   #SF_Alarm13(IB1In := NOT "STATUS_110".GM01_BG02 AND "STATUS_110".MatCard[3, 1].Occupied,   // "STD_DI_Mon"
               IB1Inv := "STDLog0",
               IB1Ack := "STATUS_Zone100".Station110_Mode.Specific.Ack,
               IB1AlmSupp := "STATUS_Zone100".Station110_Mode.Specific.AlmSupp,
               IT_OnDly := T#2s,
               XS_Parameter := "HMI_PARAM_110".Senzor_3,
               XS_Command := "HMI_CMD_110".Senzor_3,
               OS_Status => "STATUS_110".Senzor_3);
END_REGION

REGION Network 17: Alarm - Part in lift 3 position not on map
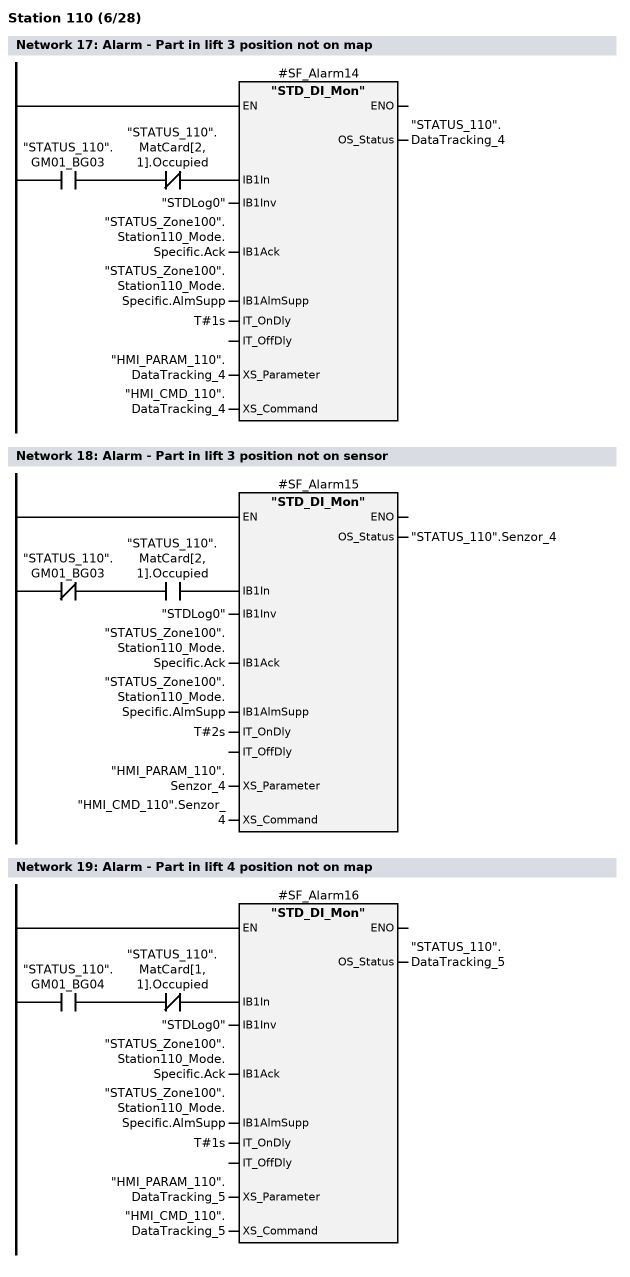
   RUNG wire#powerrail
      #SF_Alarm14(IB1In := wire#w1, IB1Inv := "STDLog0", IB1Ack := "STATUS_Zone100".Station110_Mode.Specific.Ack, IB1AlmSupp := "STATUS_Zone100".Station110_Mode.Specific.AlmSupp, IT_OnDly := T#1s, IT_OffDly :=, XS_Parameter := "HMI_PARAM_110".DataTracking_4, XS_Command := "HMI_CMD_110".DataTracking_4, OS_Status => "STATUS_110".DataTracking_4)
   END_RUNG
   RUNG wire#powerrail
      Contact( "STATUS_110".GM01_BG03 )
      I_Contact( "STATUS_110".MatCard[2, 1].Occupied )
   END_RUNG wire#w1
   // the same network as SCL:
   #SF_Alarm14(IB1In := "STATUS_110".GM01_BG03 AND NOT "STATUS_110".MatCard[2, 1].Occupied,   // "STD_DI_Mon"
               IB1Inv := "STDLog0",
               IB1Ack := "STATUS_Zone100".Station110_Mode.Specific.Ack,
               IB1AlmSupp := "STATUS_Zone100".Station110_Mode.Specific.AlmSupp,
               IT_OnDly := T#1s,
               XS_Parameter := "HMI_PARAM_110".DataTracking_4,
               XS_Command := "HMI_CMD_110".DataTracking_4,
               OS_Status => "STATUS_110".DataTracking_4);
END_REGION

REGION Network 18: Alarm - Part in lift 3 position not on sensor
   RUNG wire#powerrail
      #SF_Alarm15(IB1In := wire#w1, IB1Inv := "STDLog0", IB1Ack := "STATUS_Zone100".Station110_Mode.Specific.Ack, IB1AlmSupp := "STATUS_Zone100".Station110_Mode.Specific.AlmSupp, IT_OnDly := T#2s, IT_OffDly :=, XS_Parameter := "HMI_PARAM_110".Senzor_4, XS_Command := "HMI_CMD_110".Senzor_4, OS_Status => "STATUS_110".Senzor_4)
   END_RUNG
   RUNG wire#powerrail
      I_Contact( "STATUS_110".GM01_BG03 )
      Contact( "STATUS_110".MatCard[2, 1].Occupied )
   END_RUNG wire#w1
   // the same network as SCL:
   #SF_Alarm15(IB1In := NOT "STATUS_110".GM01_BG03 AND "STATUS_110".MatCard[2, 1].Occupied,   // "STD_DI_Mon"
               IB1Inv := "STDLog0",
               IB1Ack := "STATUS_Zone100".Station110_Mode.Specific.Ack,
               IB1AlmSupp := "STATUS_Zone100".Station110_Mode.Specific.AlmSupp,
               IT_OnDly := T#2s,
               XS_Parameter := "HMI_PARAM_110".Senzor_4,
               XS_Command := "HMI_CMD_110".Senzor_4,
               OS_Status => "STATUS_110".Senzor_4);
END_REGION

REGION Network 19: Alarm - Part in lift 4 position not on map
   RUNG wire#powerrail
      #SF_Alarm16(IB1In := wire#w1, IB1Inv := "STDLog0", IB1Ack := "STATUS_Zone100".Station110_Mode.Specific.Ack, IB1AlmSupp := "STATUS_Zone100".Station110_Mode.Specific.AlmSupp, IT_OnDly := T#1s, IT_OffDly :=, XS_Parameter := "HMI_PARAM_110".DataTracking_5, XS_Command := "HMI_CMD_110".DataTracking_5, OS_Status => "STATUS_110".DataTracking_5)
   END_RUNG
   RUNG wire#powerrail
      Contact( "STATUS_110".GM01_BG04 )
      I_Contact( "STATUS_110".MatCard[1, 1].Occupied )
   END_RUNG wire#w1
   // the same network as SCL:
   #SF_Alarm16(IB1In := "STATUS_110".GM01_BG04 AND NOT "STATUS_110".MatCard[1, 1].Occupied,   // "STD_DI_Mon"
               IB1Inv := "STDLog0",
               IB1Ack := "STATUS_Zone100".Station110_Mode.Specific.Ack,
               IB1AlmSupp := "STATUS_Zone100".Station110_Mode.Specific.AlmSupp,
               IT_OnDly := T#1s,
               XS_Parameter := "HMI_PARAM_110".DataTracking_5,
               XS_Command := "HMI_CMD_110".DataTracking_5,
               OS_Status => "STATUS_110".DataTracking_5);
END_REGION

REGION Network 20: Alarm - Part in lift 4 position not on sensor
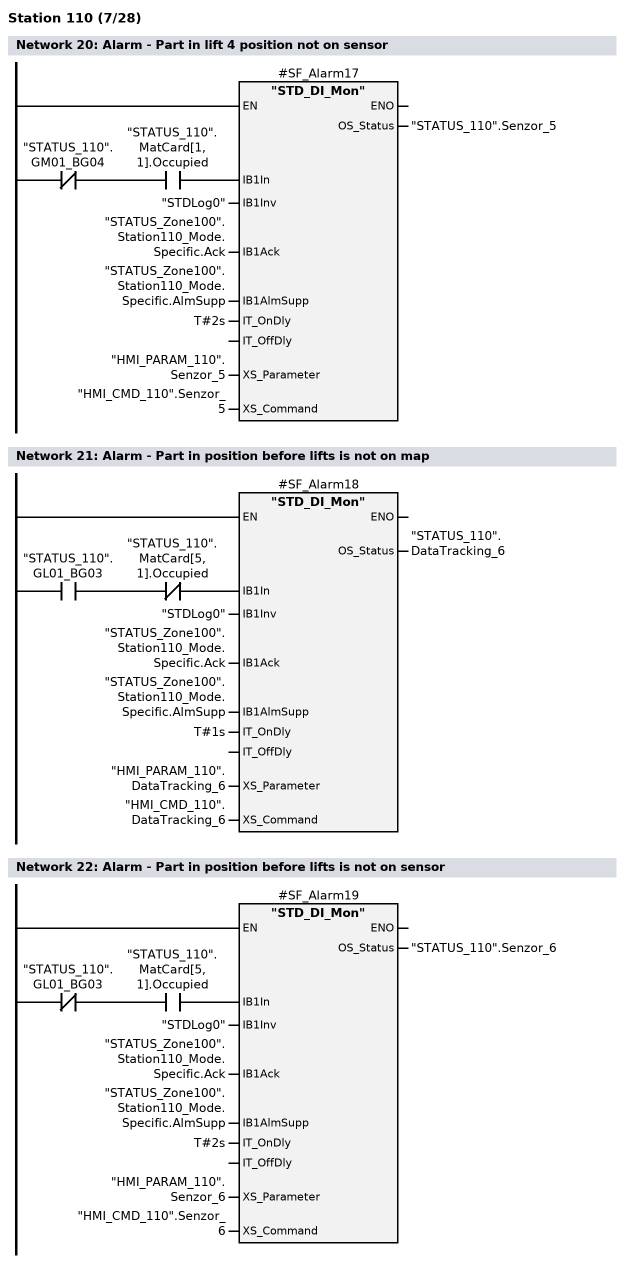
   RUNG wire#powerrail
      #SF_Alarm17(IB1In := wire#w1, IB1Inv := "STDLog0", IB1Ack := "STATUS_Zone100".Station110_Mode.Specific.Ack, IB1AlmSupp := "STATUS_Zone100".Station110_Mode.Specific.AlmSupp, IT_OnDly := T#2s, IT_OffDly :=, XS_Parameter := "HMI_PARAM_110".Senzor_5, XS_Command := "HMI_CMD_110".Senzor_5, OS_Status => "STATUS_110".Senzor_5)
   END_RUNG
   RUNG wire#powerrail
      I_Contact( "STATUS_110".GM01_BG04 )
      Contact( "STATUS_110".MatCard[1, 1].Occupied )
   END_RUNG wire#w1
   // the same network as SCL:
   #SF_Alarm17(IB1In := NOT "STATUS_110".GM01_BG04 AND "STATUS_110".MatCard[1, 1].Occupied,   // "STD_DI_Mon"
               IB1Inv := "STDLog0",
               IB1Ack := "STATUS_Zone100".Station110_Mode.Specific.Ack,
               IB1AlmSupp := "STATUS_Zone100".Station110_Mode.Specific.AlmSupp,
               IT_OnDly := T#2s,
               XS_Parameter := "HMI_PARAM_110".Senzor_5,
               XS_Command := "HMI_CMD_110".Senzor_5,
               OS_Status => "STATUS_110".Senzor_5);
END_REGION

REGION Network 21: Alarm - Part in position before lifts is not on map
   RUNG wire#powerrail
      #SF_Alarm18(IB1In := wire#w1, IB1Inv := "STDLog0", IB1Ack := "STATUS_Zone100".Station110_Mode.Specific.Ack, IB1AlmSupp := "STATUS_Zone100".Station110_Mode.Specific.AlmSupp, IT_OnDly := T#1s, IT_OffDly :=, XS_Parameter := "HMI_PARAM_110".DataTracking_6, XS_Command := "HMI_CMD_110".DataTracking_6, OS_Status => "STATUS_110".DataTracking_6)
   END_RUNG
   RUNG wire#powerrail
      Contact( "STATUS_110".GL01_BG03 )
      I_Contact( "STATUS_110".MatCard[5, 1].Occupied )
   END_RUNG wire#w1
   // the same network as SCL:
   #SF_Alarm18(IB1In := "STATUS_110".GL01_BG03 AND NOT "STATUS_110".MatCard[5, 1].Occupied,   // "STD_DI_Mon"
               IB1Inv := "STDLog0",
               IB1Ack := "STATUS_Zone100".Station110_Mode.Specific.Ack,
               IB1AlmSupp := "STATUS_Zone100".Station110_Mode.Specific.AlmSupp,
               IT_OnDly := T#1s,
               XS_Parameter := "HMI_PARAM_110".DataTracking_6,
               XS_Command := "HMI_CMD_110".DataTracking_6,
               OS_Status => "STATUS_110".DataTracking_6);
END_REGION

REGION Network 22: Alarm - Part in position before lifts is not on sensor
   RUNG wire#powerrail
      #SF_Alarm19(IB1In := wire#w1, IB1Inv := "STDLog0", IB1Ack := "STATUS_Zone100".Station110_Mode.Specific.Ack, IB1AlmSupp := "STATUS_Zone100".Station110_Mode.Specific.AlmSupp, IT_OnDly := T#2s, IT_OffDly :=, XS_Parameter := "HMI_PARAM_110".Senzor_6, XS_Command := "HMI_CMD_110".Senzor_6, OS_Status => "STATUS_110".Senzor_6)
   END_RUNG
   RUNG wire#powerrail
      I_Contact( "STATUS_110".GL01_BG03 )
      Contact( "STATUS_110".MatCard[5, 1].Occupied )
   END_RUNG wire#w1
   // the same network as SCL:
   #SF_Alarm19(IB1In := NOT "STATUS_110".GL01_BG03 AND "STATUS_110".MatCard[5, 1].Occupied,   // "STD_DI_Mon"
               IB1Inv := "STDLog0",
               IB1Ack := "STATUS_Zone100".Station110_Mode.Specific.Ack,
               IB1AlmSupp := "STATUS_Zone100".Station110_Mode.Specific.AlmSupp,
               IT_OnDly := T#2s,
               XS_Parameter := "HMI_PARAM_110".Senzor_6,
               XS_Command := "HMI_CMD_110".Senzor_6,
               OS_Status => "STATUS_110".Senzor_6);
END_REGION

REGION Network 23: Alarm - Part behind last lift
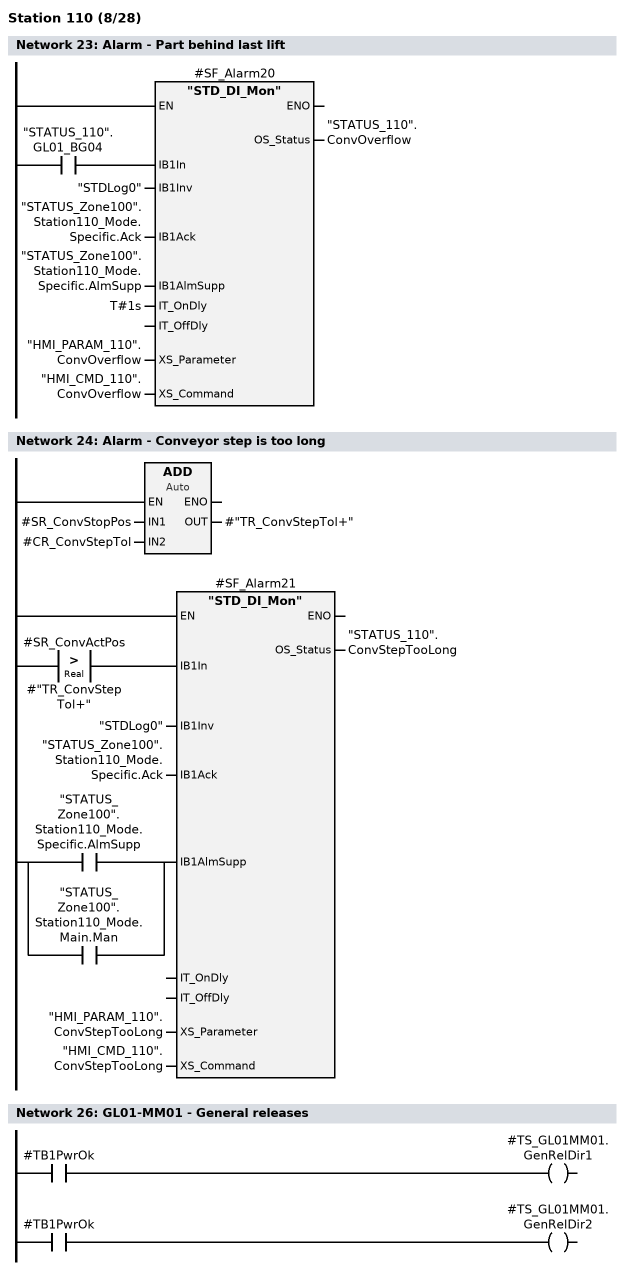
   RUNG wire#powerrail
      #SF_Alarm20(IB1In := wire#w1, IB1Inv := "STDLog0", IB1Ack := "STATUS_Zone100".Station110_Mode.Specific.Ack, IB1AlmSupp := "STATUS_Zone100".Station110_Mode.Specific.AlmSupp, IT_OnDly := T#1s, IT_OffDly :=, XS_Parameter := "HMI_PARAM_110".ConvOverflow, XS_Command := "HMI_CMD_110".ConvOverflow, OS_Status => "STATUS_110".ConvOverflow)
   END_RUNG
   RUNG wire#powerrail
      Contact( "STATUS_110".GL01_BG04 )
   END_RUNG wire#w1
   // the same network as SCL:
   #SF_Alarm20(IB1In := "STATUS_110".GL01_BG04,   // "STD_DI_Mon"
               IB1Inv := "STDLog0",
               IB1Ack := "STATUS_Zone100".Station110_Mode.Specific.Ack,
               IB1AlmSupp := "STATUS_Zone100".Station110_Mode.Specific.AlmSupp,
               IT_OnDly := T#1s,
               XS_Parameter := "HMI_PARAM_110".ConvOverflow,
               XS_Command := "HMI_CMD_110".ConvOverflow,
               OS_Status => "STATUS_110".ConvOverflow);
END_REGION

REGION Network 24: Alarm - Conveyor step is too long
   RUNG wire#powerrail
      Add(in1 := #SR_ConvStopPos, in2 := #CR_ConvStepTol, out => #"TR_ConvStepTol+")
   END_RUNG
   RUNG wire#powerrail
      #SF_Alarm21(IB1In := wire#w1, IB1AlmSupp := wire#w2, IB1Inv := "STDLog0", IB1Ack := "STATUS_Zone100".Station110_Mode.Specific.Ack, IT_OnDly :=, IT_OffDly :=, XS_Parameter := "HMI_PARAM_110".ConvStepTooLong, XS_Command := "HMI_CMD_110".ConvStepTooLong, OS_Status => "STATUS_110".ConvStepTooLong)
   END_RUNG
   RUNG wire#powerrail
      { S7_Templates := "SrcType := Real" } GT_Contact(in1 := #SR_ConvActPos, in2 := #"TR_ConvStepTol+")
   END_RUNG wire#w1
   RUNG wire#powerrail
      Contact( "STATUS_Zone100".Station110_Mode.Specific.AlmSupp )
   END_RUNG wire#w2
   RUNG wire#powerrail
      Contact( "STATUS_Zone100".Station110_Mode.Main.Man )
   END_RUNG wire#w2
   // the same network as SCL:
   #"TR_ConvStepTol+" := #SR_ConvStopPos + #CR_ConvStepTol;
   #SF_Alarm21(IB1In := #SR_ConvActPos > #"TR_ConvStepTol+",   // "STD_DI_Mon"
               IB1Inv := "STDLog0",
               IB1Ack := "STATUS_Zone100".Station110_Mode.Specific.Ack,
               IB1AlmSupp := "STATUS_Zone100".Station110_Mode.Specific.AlmSupp OR "STATUS_Zone100".Station110_Mode.Main.Man,
               XS_Parameter := "HMI_PARAM_110".ConvStepTooLong,
               XS_Command := "HMI_CMD_110".ConvStepTooLong,
               OS_Status => "STATUS_110".ConvStepTooLong);
END_REGION

REGION Network 25: *************** GL01-MM01 - Stopper ***************
END_REGION

REGION Network 26: GL01-MM01 - General releases
   RUNG wire#powerrail
      Contact( #TB1PwrOk )
      Coil( #TS_GL01MM01.GenRelDir1 )
   END_RUNG
   RUNG wire#powerrail
      Contact( #TB1PwrOk )
      Coil( #TS_GL01MM01.GenRelDir2 )
   END_RUNG
   // the same network as SCL:
   #TS_GL01MM01.GenRelDir1 := #TB1PwrOk;
   #TS_GL01MM01.GenRelDir2 := #TB1PwrOk;
END_REGION

REGION Network 27: GL01-MM01 - Interlocks
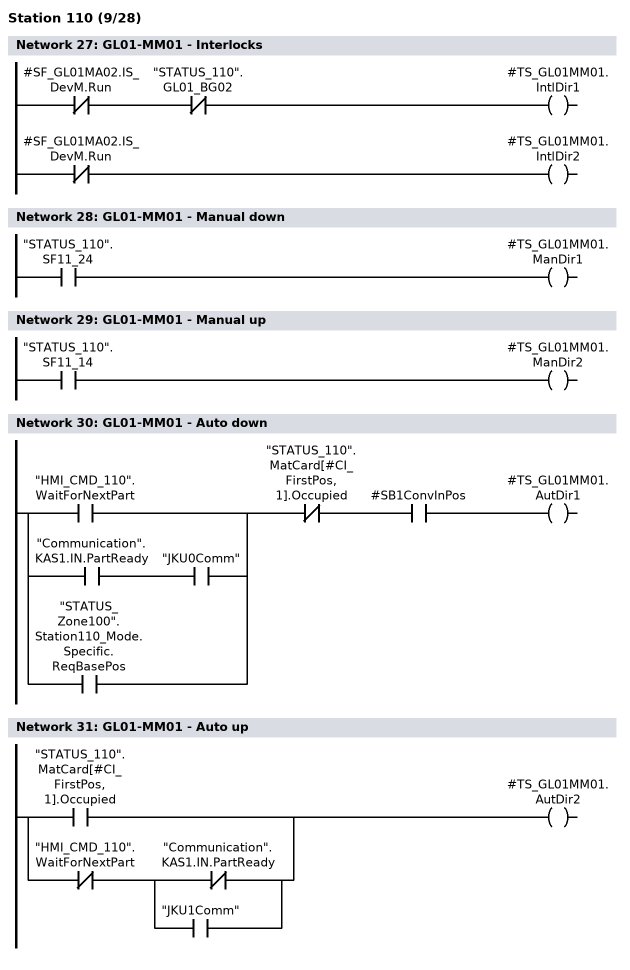
   RUNG wire#powerrail
      I_Contact( #SF_GL01MA02.IS_DevM.Run )
      I_Contact( "STATUS_110".GL01_BG02 )
      Coil( #TS_GL01MM01.IntlDir1 )
   END_RUNG
   RUNG wire#powerrail
      I_Contact( #SF_GL01MA02.IS_DevM.Run )
      Coil( #TS_GL01MM01.IntlDir2 )
   END_RUNG
   // the same network as SCL:
   #TS_GL01MM01.IntlDir1 := NOT #SF_GL01MA02.IS_DevM.Run AND NOT "STATUS_110".GL01_BG02;
   #TS_GL01MM01.IntlDir2 := NOT #SF_GL01MA02.IS_DevM.Run;
END_REGION

REGION Network 28: GL01-MM01 - Manual down
   RUNG wire#powerrail
      Contact( "STATUS_110".SF11_24 )
      Coil( #TS_GL01MM01.ManDir1 )
   END_RUNG
   // the same network as SCL:
   #TS_GL01MM01.ManDir1 := "STATUS_110".SF11_24;
END_REGION

REGION Network 29: GL01-MM01 - Manual up
   RUNG wire#powerrail
      Contact( "STATUS_110".SF11_14 )
      Coil( #TS_GL01MM01.ManDir2 )
   END_RUNG
   // the same network as SCL:
   #TS_GL01MM01.ManDir2 := "STATUS_110".SF11_14;
END_REGION

REGION Network 30: GL01-MM01 - Auto down
   RUNG wire#powerrail
      Contact( "HMI_CMD_110".WaitForNextPart )
      wire#w1
      I_Contact( "STATUS_110".MatCard[#CI_FirstPos, 1].Occupied )
      Contact( #SB1ConvInPos )
      Coil( #TS_GL01MM01.AutDir1 )
   END_RUNG
   RUNG wire#powerrail
      Contact( "Communication".KAS1.IN.PartReady )
      Contact( "JKU0Comm" )
   END_RUNG wire#w1
   RUNG wire#powerrail
      Contact( "STATUS_Zone100".Station110_Mode.Specific.ReqBasePos )
   END_RUNG wire#w1
   // the same network as SCL:
   #TS_GL01MM01.AutDir1 := ("HMI_CMD_110".WaitForNextPart OR ("Communication".KAS1.IN.PartReady AND "JKU0Comm") OR "STATUS_Zone100".Station110_Mode.Specific.ReqBasePos) AND NOT "STATUS_110".MatCard[#CI_FirstPos, 1].Occupied AND #SB1ConvInPos;
END_REGION

REGION Network 31: GL01-MM01 - Auto up
   RUNG wire#powerrail
      Contact( "STATUS_110".MatCard[#CI_FirstPos, 1].Occupied )
      wire#w1
      Coil( #TS_GL01MM01.AutDir2 )
   END_RUNG
   RUNG wire#powerrail
      I_Contact( "HMI_CMD_110".WaitForNextPart )
      wire#w2
      I_Contact( "Communication".KAS1.IN.PartReady )
   END_RUNG wire#w1
   RUNG wire#w2
      Contact( "JKU1Comm" )
   END_RUNG wire#w1
   // the same network as SCL:
   #TS_GL01MM01.AutDir2 := "STATUS_110".MatCard[#CI_FirstPos, 1].Occupied OR (NOT "HMI_CMD_110".WaitForNextPart AND (NOT "Communication".KAS1.IN.PartReady OR "JKU1Comm"));
END_REGION

REGION Network 32: GL01-MM01 - Valve control
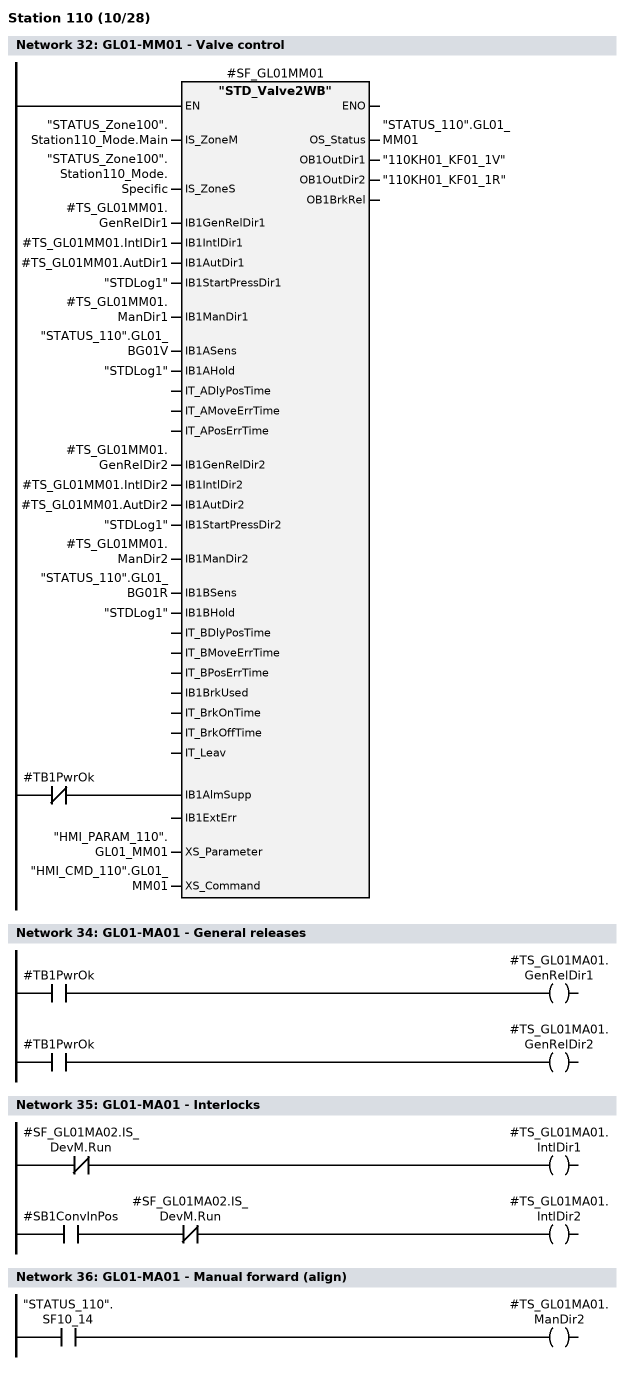
   RUNG wire#powerrail
      #SF_GL01MM01(IB1AlmSupp := wire#w1, IS_ZoneM := "STATUS_Zone100".Station110_Mode.Main, IS_ZoneS := "STATUS_Zone100".Station110_Mode.Specific, IB1GenRelDir1 := #TS_GL01MM01.GenRelDir1, IB1IntlDir1 := #TS_GL01MM01.IntlDir1, IB1AutDir1 := #TS_GL01MM01.AutDir1, IB1StartPressDir1 := "STDLog1", IB1ManDir1 := #TS_GL01MM01.ManDir1, IB1ASens := "STATUS_110".GL01_BG01V, IB1AHold := "STDLog1", IT_ADlyPosTime :=, IT_AMoveErrTime :=, IT_APosErrTime :=, IB1GenRelDir2 := #TS_GL01MM01.GenRelDir2, IB1IntlDir2 := #TS_GL01MM01.IntlDir2, IB1AutDir2 := #TS_GL01MM01.AutDir2, IB1StartPressDir2 := "STDLog1", IB1ManDir2 := #TS_GL01MM01.ManDir2, IB1BSens := "STATUS_110".GL01_BG01R, IB1BHold := "STDLog1", IT_BDlyPosTime :=, IT_BMoveErrTime :=, IT_BPosErrTime :=, IB1BrkUsed :=, IT_BrkOnTime :=, IT_BrkOffTime :=, IT_Leav :=, IB1ExtErr :=, XS_Parameter := "HMI_PARAM_110".GL01_MM01, XS_Command := "HMI_CMD_110".GL01_MM01, OS_Status => "STATUS_110".GL01_MM01, OB1OutDir1 => "110KH01_KF01_1V", OB1OutDir2 => "110KH01_KF01_1R", OB1BrkRel =>)
   END_RUNG
   RUNG wire#powerrail
      I_Contact( #TB1PwrOk )
   END_RUNG wire#w1
   // the same network as SCL:
   #SF_GL01MM01(IS_ZoneM := "STATUS_Zone100".Station110_Mode.Main,   // "STD_Valve2WB"
                IS_ZoneS := "STATUS_Zone100".Station110_Mode.Specific,
                IB1GenRelDir1 := #TS_GL01MM01.GenRelDir1,
                IB1IntlDir1 := #TS_GL01MM01.IntlDir1,
                IB1AutDir1 := #TS_GL01MM01.AutDir1,
                IB1StartPressDir1 := "STDLog1",
                IB1ManDir1 := #TS_GL01MM01.ManDir1,
                IB1ASens := "STATUS_110".GL01_BG01V,
                IB1AHold := "STDLog1",
                IB1GenRelDir2 := #TS_GL01MM01.GenRelDir2,
                IB1IntlDir2 := #TS_GL01MM01.IntlDir2,
                IB1AutDir2 := #TS_GL01MM01.AutDir2,
                IB1StartPressDir2 := "STDLog1",
                IB1ManDir2 := #TS_GL01MM01.ManDir2,
                IB1BSens := "STATUS_110".GL01_BG01R,
                IB1BHold := "STDLog1",
                IB1AlmSupp := NOT #TB1PwrOk,
                XS_Parameter := "HMI_PARAM_110".GL01_MM01,
                XS_Command := "HMI_CMD_110".GL01_MM01,
                OS_Status => "STATUS_110".GL01_MM01,
                OB1OutDir1 => "110KH01_KF01_1V",
                OB1OutDir2 => "110KH01_KF01_1R");
END_REGION

REGION Network 33: *************** GL01-MA01 - Part aligner ***************
   // Axis range - 0...600 mm
END_REGION

REGION Network 34: GL01-MA01 - General releases
   RUNG wire#powerrail
      Contact( #TB1PwrOk )
      Coil( #TS_GL01MA01.GenRelDir1 )
   END_RUNG
   RUNG wire#powerrail
      Contact( #TB1PwrOk )
      Coil( #TS_GL01MA01.GenRelDir2 )
   END_RUNG
   // the same network as SCL:
   #TS_GL01MA01.GenRelDir1 := #TB1PwrOk;
   #TS_GL01MA01.GenRelDir2 := #TB1PwrOk;
END_REGION

REGION Network 35: GL01-MA01 - Interlocks
   RUNG wire#powerrail
      I_Contact( #SF_GL01MA02.IS_DevM.Run )
      Coil( #TS_GL01MA01.IntlDir1 )
   END_RUNG
   RUNG wire#powerrail
      Contact( #SB1ConvInPos )
      I_Contact( #SF_GL01MA02.IS_DevM.Run )
      Coil( #TS_GL01MA01.IntlDir2 )
   END_RUNG
   // the same network as SCL:
   #TS_GL01MA01.IntlDir1 := NOT #SF_GL01MA02.IS_DevM.Run;
   #TS_GL01MA01.IntlDir2 := #SB1ConvInPos AND NOT #SF_GL01MA02.IS_DevM.Run;
END_REGION

REGION Network 36: GL01-MA01 - Manual forward (align)
   RUNG wire#powerrail
      Contact( "STATUS_110".SF10_14 )
      Coil( #TS_GL01MA01.ManDir2 )
   END_RUNG
   // the same network as SCL:
   #TS_GL01MA01.ManDir2 := "STATUS_110".SF10_14;
END_REGION

REGION Network 37: GL01-MA01 - Manual backward (return)
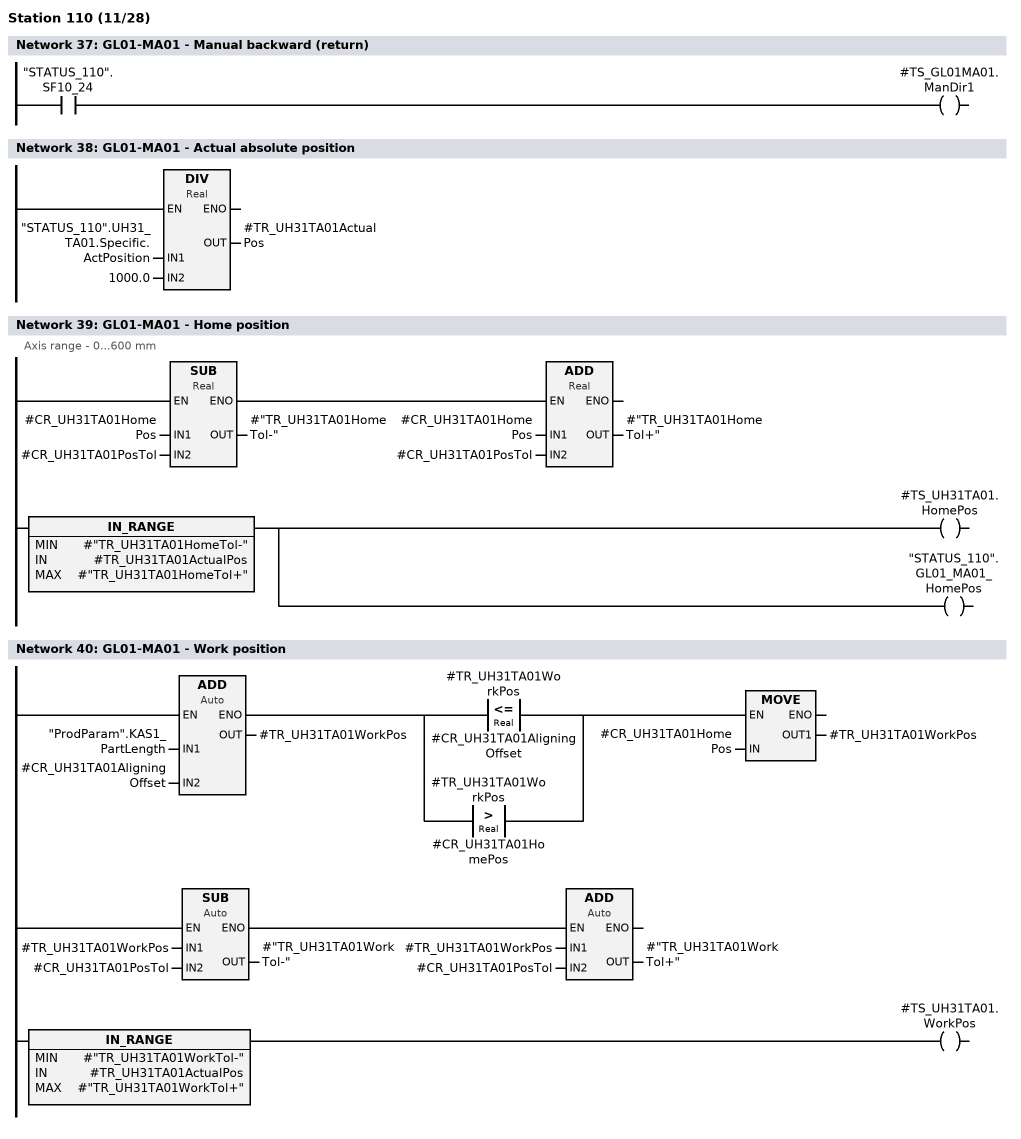
   RUNG wire#powerrail
      Contact( "STATUS_110".SF10_24 )
      Coil( #TS_GL01MA01.ManDir1 )
   END_RUNG
   // the same network as SCL:
   #TS_GL01MA01.ManDir1 := "STATUS_110".SF10_24;
END_REGION

REGION Network 38: GL01-MA01 - Actual absolute position
   RUNG wire#powerrail
      { S7_Templates := "SrcType := Real" } Div(in1 := "STATUS_110".UH31_TA01.Specific.ActPosition, in2 := 1000.0, out => #TR_UH31TA01ActualPos)
   END_RUNG
   // the same network as SCL:
   #TR_UH31TA01ActualPos := "STATUS_110".UH31_TA01.Specific.ActPosition / 1000.0;
END_REGION

REGION Network 39: GL01-MA01 - Home position
   // Axis range - 0...600 mm
   RUNG wire#powerrail
      { S7_Templates := "SrcType := Real" } Sub(in1 := #CR_UH31TA01HomePos, in2 := #CR_UH31TA01PosTol, out => #"TR_UH31TA01HomeTol-")
      { S7_Templates := "SrcType := Real" } Add(in1 := #CR_UH31TA01HomePos, in2 := #CR_UH31TA01PosTol, out => #"TR_UH31TA01HomeTol+")
   END_RUNG
   RUNG wire#powerrail
      { S7_Templates := "SrcType := Real" } InRange(min := #"TR_UH31TA01HomeTol-", in := #TR_UH31TA01ActualPos, max := #"TR_UH31TA01HomeTol+")
      wire#w1
      Coil( #TS_UH31TA01.HomePos )
   END_RUNG
   RUNG wire#w1
      Coil( "STATUS_110".GL01_MA01_HomePos )
   END_RUNG
   // the same network as SCL:
   #"TR_UH31TA01HomeTol-" := #CR_UH31TA01HomePos - #CR_UH31TA01PosTol;
   #"TR_UH31TA01HomeTol+" := #CR_UH31TA01HomePos + #CR_UH31TA01PosTol;
   #TS_UH31TA01.HomePos := (#"TR_UH31TA01HomeTol-" <= #TR_UH31TA01ActualPos) AND (#TR_UH31TA01ActualPos <= #"TR_UH31TA01HomeTol+");
   "STATUS_110".GL01_MA01_HomePos := #TS_UH31TA01.HomePos;
END_REGION

REGION Network 40: GL01-MA01 - Work position
   RUNG wire#powerrail
      Add(in1 := "ProdParam".KAS1_PartLength, in2 := #CR_UH31TA01AligningOffset, out => #TR_UH31TA01WorkPos)
      wire#w1
      { S7_Templates := "SrcType := Real" } LE_Contact(in1 := #TR_UH31TA01WorkPos, in2 := #CR_UH31TA01AligningOffset)
      wire#w2
      Move(in := #CR_UH31TA01HomePos, out1 => #TR_UH31TA01WorkPos)
   END_RUNG
   RUNG wire#w1
      { S7_Templates := "SrcType := Real" } GT_Contact(in1 := #TR_UH31TA01WorkPos, in2 := #CR_UH31TA01HomePos)
   END_RUNG wire#w2
   RUNG wire#powerrail
      Sub(in1 := #TR_UH31TA01WorkPos, in2 := #CR_UH31TA01PosTol, out => #"TR_UH31TA01WorkTol-")
      Add(in1 := #TR_UH31TA01WorkPos, in2 := #CR_UH31TA01PosTol, out => #"TR_UH31TA01WorkTol+")
   END_RUNG
   RUNG wire#powerrail
      { S7_Templates := "SrcType := Real" } InRange(min := #"TR_UH31TA01WorkTol-", in := #TR_UH31TA01ActualPos, max := #"TR_UH31TA01WorkTol+")
      Coil( #TS_UH31TA01.WorkPos )
   END_RUNG
   // the same network as SCL:
   #TR_UH31TA01WorkPos := "ProdParam".KAS1_PartLength + #CR_UH31TA01AligningOffset;
   IF (#TR_UH31TA01WorkPos <= #CR_UH31TA01AligningOffset) OR (#TR_UH31TA01WorkPos > #CR_UH31TA01HomePos) THEN
       #TR_UH31TA01WorkPos := #CR_UH31TA01HomePos;
   END_IF;
   #"TR_UH31TA01WorkTol-" := #TR_UH31TA01WorkPos - #CR_UH31TA01PosTol;
   #"TR_UH31TA01WorkTol+" := #TR_UH31TA01WorkPos + #CR_UH31TA01PosTol;
   #TS_UH31TA01.WorkPos := (#"TR_UH31TA01WorkTol-" <= #TR_UH31TA01ActualPos) AND (#TR_UH31TA01ActualPos <= #"TR_UH31TA01WorkTol+");
END_REGION

REGION Network 41: GL01-MA01 - Enable work
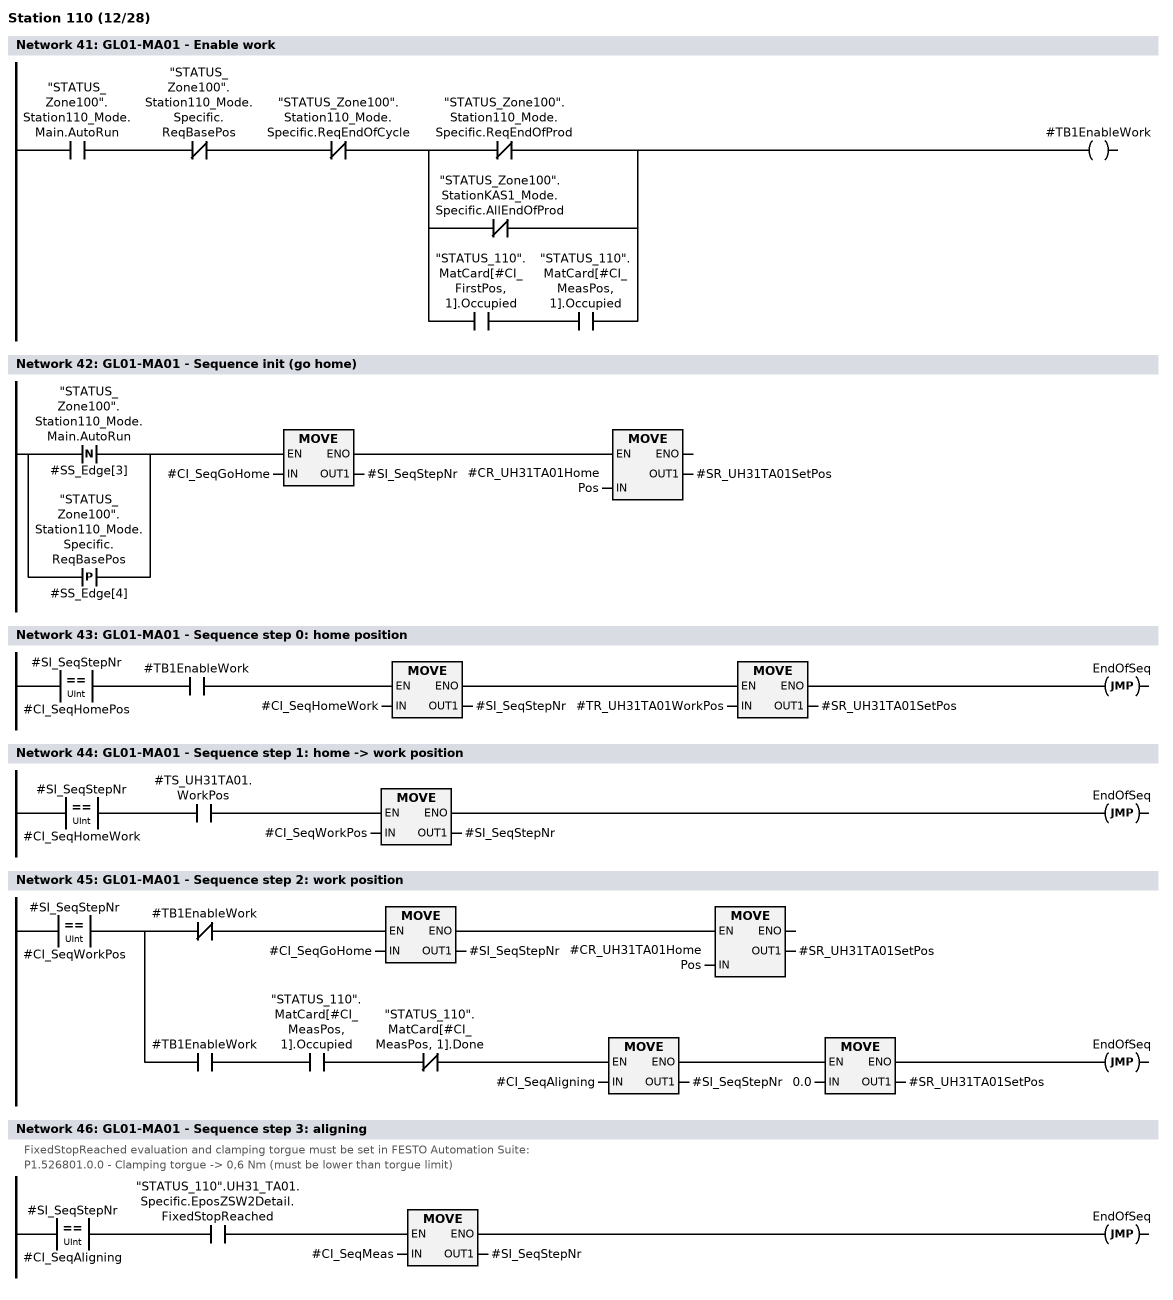
   RUNG wire#powerrail
      Contact( "STATUS_Zone100".Station110_Mode.Main.AutoRun )
      I_Contact( "STATUS_Zone100".Station110_Mode.Specific.ReqBasePos )
      I_Contact( "STATUS_Zone100".Station110_Mode.Specific.ReqEndOfCycle )
      wire#w1
      I_Contact( "STATUS_Zone100".Station110_Mode.Specific.ReqEndOfProd )
      wire#w2
      Coil( #TB1EnableWork )
   END_RUNG
   RUNG wire#w1
      I_Contact( "STATUS_Zone100".StationKAS1_Mode.Specific.AllEndOfProd )
   END_RUNG wire#w2
   RUNG wire#w1
      Contact( "STATUS_110".MatCard[#CI_FirstPos, 1].Occupied )
      Contact( "STATUS_110".MatCard[#CI_MeasPos, 1].Occupied )
   END_RUNG wire#w2
   // the same network as SCL:
   #TB1EnableWork := "STATUS_Zone100".Station110_Mode.Main.AutoRun AND NOT "STATUS_Zone100".Station110_Mode.Specific.ReqBasePos AND NOT "STATUS_Zone100".Station110_Mode.Specific.ReqEndOfCycle AND (NOT "STATUS_Zone100".Station110_Mode.Specific.ReqEndOfProd OR NOT "STATUS_Zone100".StationKAS1_Mode.Specific.AllEndOfProd OR ("STATUS_110".MatCard[#CI_FirstPos, 1].Occupied AND "STATUS_110".MatCard[#CI_MeasPos, 1].Occupied));
END_REGION

REGION Network 42: GL01-MA01 - Sequence init (go home)
   RUNG wire#powerrail
      N_Contact(operand := "STATUS_Zone100".Station110_Mode.Main.AutoRun, bit := #SS_Edge[3])
      wire#w1
      Move(in := #CI_SeqGoHome, out1 => #SI_SeqStepNr)
      Move(in := #CR_UH31TA01HomePos, out1 => #SR_UH31TA01SetPos)
   END_RUNG
   RUNG wire#powerrail
      P_Contact(operand := "STATUS_Zone100".Station110_Mode.Specific.ReqBasePos, bit := #SS_Edge[4])
   END_RUNG wire#w1
   // the same network as SCL:
   #_w1 := NOT "STATUS_Zone100".Station110_Mode.Main.AutoRun AND #SS_Edge[3];   // falling edge of "STATUS_Zone100".Station110_Mode.Main.AutoRun
   #SS_Edge[3] := "STATUS_Zone100".Station110_Mode.Main.AutoRun;
   #_w2 := "STATUS_Zone100".Station110_Mode.Specific.ReqBasePos AND NOT #SS_Edge[4];   // rising edge of "STATUS_Zone100".Station110_Mode.Specific.ReqBasePos
   #SS_Edge[4] := "STATUS_Zone100".Station110_Mode.Specific.ReqBasePos;
   IF #_w1 OR #_w2 THEN
       #SI_SeqStepNr := #CI_SeqGoHome;
       #SR_UH31TA01SetPos := #CR_UH31TA01HomePos;
   END_IF;
END_REGION

REGION Network 43: GL01-MA01 - Sequence step 0: home position
   RUNG wire#powerrail
      { S7_Templates := "SrcType := UInt" } EQ_Contact(in1 := #SI_SeqStepNr, in2 := #CI_SeqHomePos)
      Contact( #TB1EnableWork )
      Move(in := #CI_SeqHomeWork, out1 => #SI_SeqStepNr)
      Move(in := #TR_UH31TA01WorkPos, out1 => #SR_UH31TA01SetPos)
      JumpCoil( EndOfSeq )
   END_RUNG
   // the same network as SCL:
   #_w1 := (#SI_SeqStepNr = #CI_SeqHomePos) AND #TB1EnableWork;
   IF #_w1 THEN
       #SI_SeqStepNr := #CI_SeqHomeWork;
       #SR_UH31TA01SetPos := #TR_UH31TA01WorkPos;
       GOTO EndOfSeq;
   END_IF;
END_REGION

REGION Network 44: GL01-MA01 - Sequence step 1: home -> work position
   RUNG wire#powerrail
      { S7_Templates := "SrcType := UInt" } EQ_Contact(in1 := #SI_SeqStepNr, in2 := #CI_SeqHomeWork)
      Contact( #TS_UH31TA01.WorkPos )
      Move(in := #CI_SeqWorkPos, out1 => #SI_SeqStepNr)
      JumpCoil( EndOfSeq )
   END_RUNG
   // the same network as SCL:
   #_w1 := (#SI_SeqStepNr = #CI_SeqHomeWork) AND #TS_UH31TA01.WorkPos;
   IF #_w1 THEN
       #SI_SeqStepNr := #CI_SeqWorkPos;
       GOTO EndOfSeq;
   END_IF;
END_REGION

REGION Network 45: GL01-MA01 - Sequence step 2: work position
   RUNG wire#powerrail
      { S7_Templates := "SrcType := UInt" } EQ_Contact(in1 := #SI_SeqStepNr, in2 := #CI_SeqWorkPos)
      wire#w1
      I_Contact( #TB1EnableWork )
      Move(in := #CI_SeqGoHome, out1 => #SI_SeqStepNr)
      Move(in := #CR_UH31TA01HomePos, out1 => #SR_UH31TA01SetPos)
   END_RUNG
   RUNG wire#w1
      Contact( #TB1EnableWork )
      Contact( "STATUS_110".MatCard[#CI_MeasPos, 1].Occupied )
      I_Contact( "STATUS_110".MatCard[#CI_MeasPos, 1].Done )
      Move(in := #CI_SeqAligning, out1 => #SI_SeqStepNr)
      Move(in := 0.0, out1 => #SR_UH31TA01SetPos)
      JumpCoil( EndOfSeq )
   END_RUNG
   // the same network as SCL:
   #_w1 := #SI_SeqStepNr = #CI_SeqWorkPos;
   IF #_w1 AND NOT #TB1EnableWork THEN
       #SI_SeqStepNr := #CI_SeqGoHome;
       #SR_UH31TA01SetPos := #CR_UH31TA01HomePos;
   END_IF;
   #_w2 := #_w1 AND #TB1EnableWork AND "STATUS_110".MatCard[#CI_MeasPos, 1].Occupied AND NOT "STATUS_110".MatCard[#CI_MeasPos, 1].Done;
   IF #_w2 THEN
       #SI_SeqStepNr := #CI_SeqAligning;
       #SR_UH31TA01SetPos := 0.0;
       GOTO EndOfSeq;
   END_IF;
END_REGION

REGION Network 46: GL01-MA01 - Sequence step 3: aligning
   // FixedStopReached evaluation and clamping torgue must be set in FESTO Automation Suite:
   // P1.526801.0.0 - Clamping torgue -> 0,6 Nm (must be lower than torgue limit)
   RUNG wire#powerrail
      { S7_Templates := "SrcType := UInt" } EQ_Contact(in1 := #SI_SeqStepNr, in2 := #CI_SeqAligning)
      Contact( "STATUS_110".UH31_TA01.Specific.EposZSW2Detail.FixedStopReached )
      Move(in := #CI_SeqMeas, out1 => #SI_SeqStepNr)
      JumpCoil( EndOfSeq )
   END_RUNG
   // the same network as SCL:
   #_w1 := (#SI_SeqStepNr = #CI_SeqAligning) AND "STATUS_110".UH31_TA01.Specific.EposZSW2Detail.FixedStopReached;
   IF #_w1 THEN
       #SI_SeqStepNr := #CI_SeqMeas;
       GOTO EndOfSeq;
   END_IF;
END_REGION

REGION Network 47: GL01-MA01 - Sequence step 4: measuring
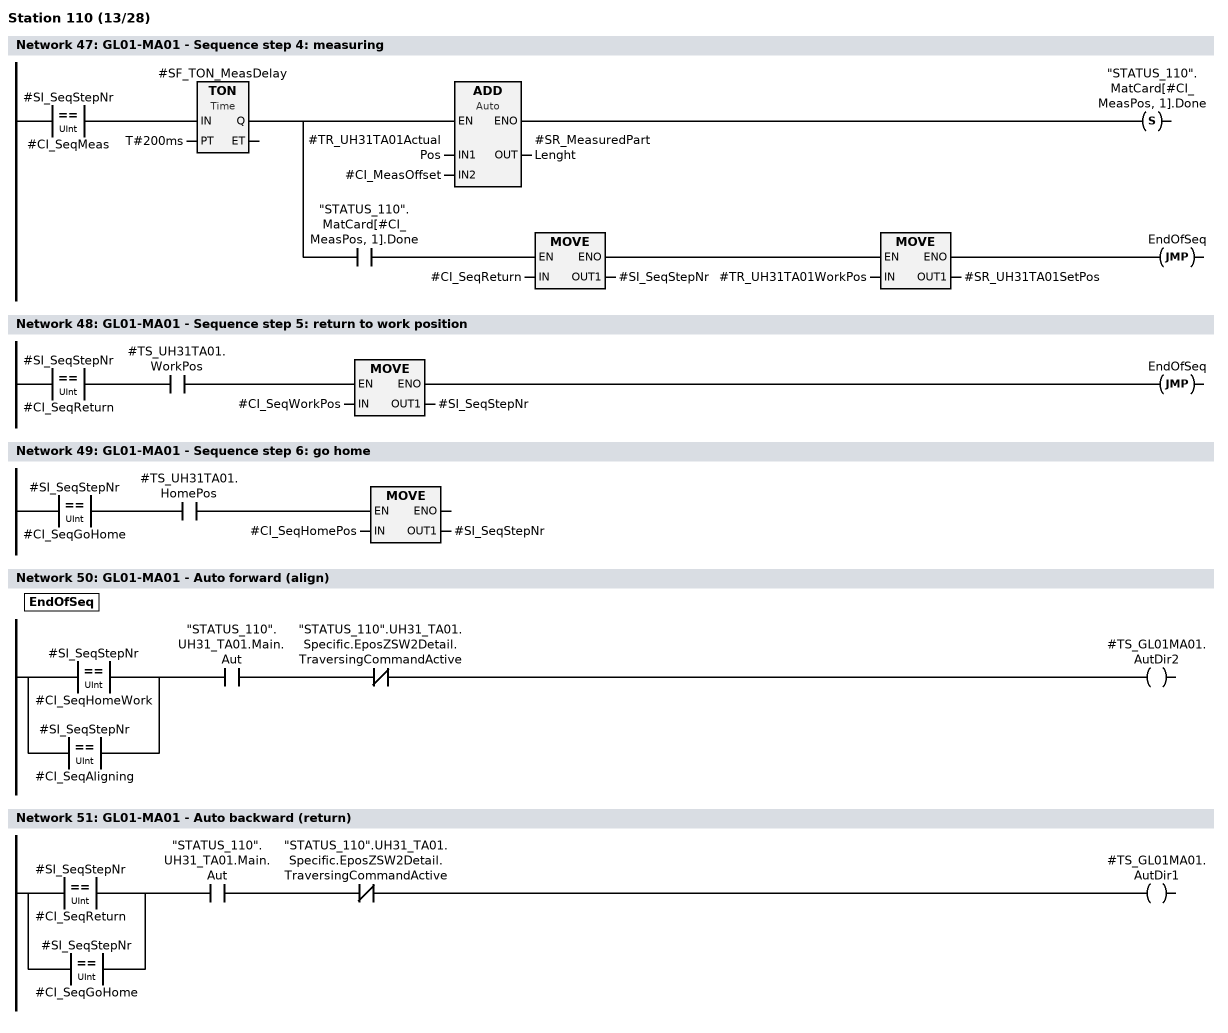
   RUNG wire#powerrail
      { S7_Templates := "SrcType := UInt" } EQ_Contact(in1 := #SI_SeqStepNr, in2 := #CI_SeqMeas)
      { S7_Templates := "time_type := Time" } #SF_TON_MeasDelay.TON(pt := T#200ms, et =>)
      wire#w1
      Add(in1 := #TR_UH31TA01ActualPos, in2 := #CI_MeasOffset, out => #SR_MeasuredPartLenght)
      S_Coil( "STATUS_110".MatCard[#CI_MeasPos, 1].Done )
   END_RUNG
   RUNG wire#w1
      Contact( "STATUS_110".MatCard[#CI_MeasPos, 1].Done )
      Move(in := #CI_SeqReturn, out1 => #SI_SeqStepNr)
      Move(in := #TR_UH31TA01WorkPos, out1 => #SR_UH31TA01SetPos)
      JumpCoil( EndOfSeq )
   END_RUNG
   // the same network as SCL:
   #SF_TON_MeasDelay(IN := #SI_SeqStepNr = #CI_SeqMeas, PT := T#200ms);   // TON
   IF #SF_TON_MeasDelay.Q THEN
       #SR_MeasuredPartLenght := #TR_UH31TA01ActualPos + #CI_MeasOffset;
       "STATUS_110".MatCard[#CI_MeasPos, 1].Done := TRUE;
   END_IF;
   #_w1 := #SF_TON_MeasDelay.Q AND "STATUS_110".MatCard[#CI_MeasPos, 1].Done;
   IF #_w1 THEN
       #SI_SeqStepNr := #CI_SeqReturn;
       #SR_UH31TA01SetPos := #TR_UH31TA01WorkPos;
       GOTO EndOfSeq;
   END_IF;
END_REGION

REGION Network 48: GL01-MA01 - Sequence step 5: return to work position
   RUNG wire#powerrail
      { S7_Templates := "SrcType := UInt" } EQ_Contact(in1 := #SI_SeqStepNr, in2 := #CI_SeqReturn)
      Contact( #TS_UH31TA01.WorkPos )
      Move(in := #CI_SeqWorkPos, out1 => #SI_SeqStepNr)
      JumpCoil( EndOfSeq )
   END_RUNG
   // the same network as SCL:
   #_w1 := (#SI_SeqStepNr = #CI_SeqReturn) AND #TS_UH31TA01.WorkPos;
   IF #_w1 THEN
       #SI_SeqStepNr := #CI_SeqWorkPos;
       GOTO EndOfSeq;
   END_IF;
END_REGION

REGION Network 49: GL01-MA01 - Sequence step 6: go home
   RUNG wire#powerrail
      { S7_Templates := "SrcType := UInt" } EQ_Contact(in1 := #SI_SeqStepNr, in2 := #CI_SeqGoHome)
      Contact( #TS_UH31TA01.HomePos )
      Move(in := #CI_SeqHomePos, out1 => #SI_SeqStepNr)
   END_RUNG
   // the same network as SCL:
   IF (#SI_SeqStepNr = #CI_SeqGoHome) AND #TS_UH31TA01.HomePos THEN #SI_SeqStepNr := #CI_SeqHomePos; END_IF;
END_REGION

REGION Network 50: GL01-MA01 - Auto forward (align)
   Label( EndOfSeq )
   RUNG wire#powerrail
      { S7_Templates := "SrcType := UInt" } EQ_Contact(in1 := #SI_SeqStepNr, in2 := #CI_SeqHomeWork)
      wire#w1
      Contact( "STATUS_110".UH31_TA01.Main.Aut )
      I_Contact( "STATUS_110".UH31_TA01.Specific.EposZSW2Detail.TraversingCommandActive )
      Coil( #TS_GL01MA01.AutDir2 )
   END_RUNG
   RUNG wire#powerrail
      { S7_Templates := "SrcType := UInt" } EQ_Contact(in1 := #SI_SeqStepNr, in2 := #CI_SeqAligning)
   END_RUNG wire#w1
   // the same network as SCL:
   EndOfSeq:
   #TS_GL01MA01.AutDir2 := ((#SI_SeqStepNr = #CI_SeqHomeWork) OR (#SI_SeqStepNr = #CI_SeqAligning)) AND "STATUS_110".UH31_TA01.Main.Aut AND NOT "STATUS_110".UH31_TA01.Specific.EposZSW2Detail.TraversingCommandActive;
END_REGION

REGION Network 51: GL01-MA01 - Auto backward (return)
   RUNG wire#powerrail
      { S7_Templates := "SrcType := UInt" } EQ_Contact(in1 := #SI_SeqStepNr, in2 := #CI_SeqReturn)
      wire#w1
      Contact( "STATUS_110".UH31_TA01.Main.Aut )
      I_Contact( "STATUS_110".UH31_TA01.Specific.EposZSW2Detail.TraversingCommandActive )
      Coil( #TS_GL01MA01.AutDir1 )
   END_RUNG
   RUNG wire#powerrail
      { S7_Templates := "SrcType := UInt" } EQ_Contact(in1 := #SI_SeqStepNr, in2 := #CI_SeqGoHome)
   END_RUNG wire#w1
   // the same network as SCL:
   #TS_GL01MA01.AutDir1 := ((#SI_SeqStepNr = #CI_SeqReturn) OR (#SI_SeqStepNr = #CI_SeqGoHome)) AND "STATUS_110".UH31_TA01.Main.Aut AND NOT "STATUS_110".UH31_TA01.Specific.EposZSW2Detail.TraversingCommandActive;
END_REGION

REGION Network 52: UH31-TA01 - FESTO servo - Set mode
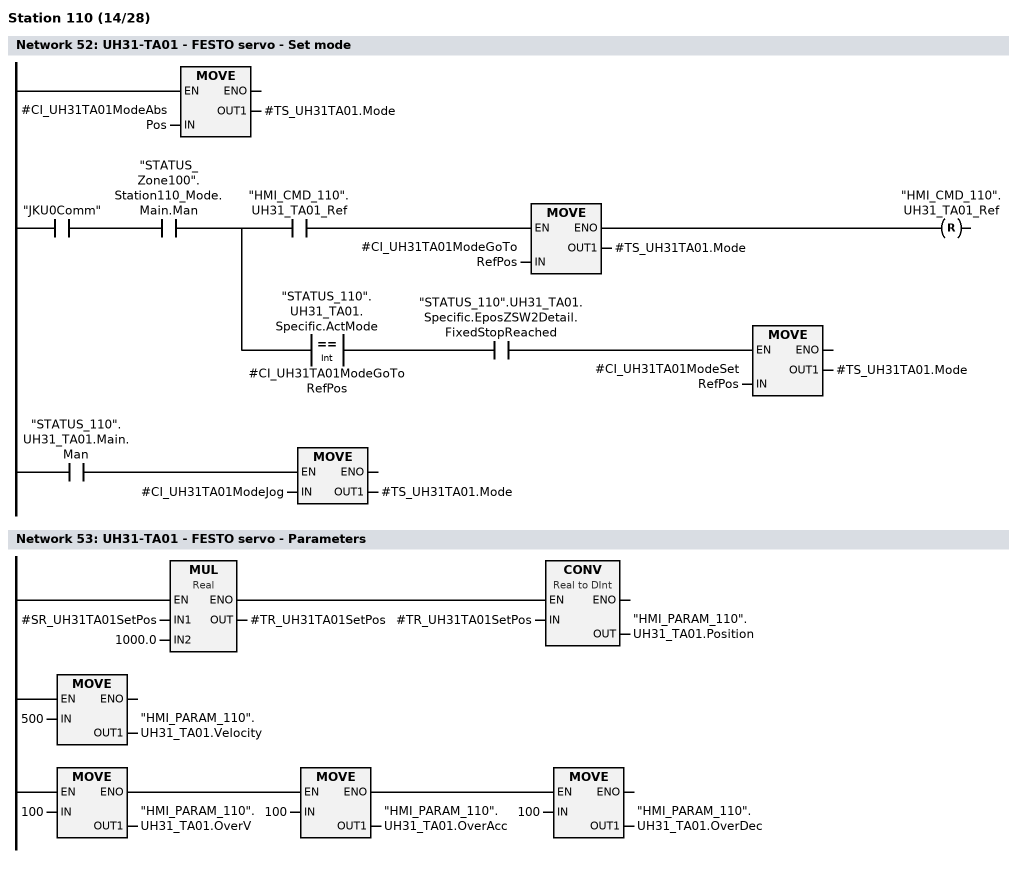
   RUNG wire#powerrail
      Move(in := #CI_UH31TA01ModeAbsPos, out1 => #TS_UH31TA01.Mode)
   END_RUNG
   RUNG wire#powerrail
      Contact( "JKU0Comm" )
      Contact( "STATUS_Zone100".Station110_Mode.Main.Man )
      wire#w1
      Contact( "HMI_CMD_110".UH31_TA01_Ref )
      Move(in := #CI_UH31TA01ModeGoToRefPos, out1 => #TS_UH31TA01.Mode)
      R_Coil( "HMI_CMD_110".UH31_TA01_Ref )
   END_RUNG
   RUNG wire#w1
      { S7_Templates := "SrcType := Int" } EQ_Contact(in1 := "STATUS_110".UH31_TA01.Specific.ActMode, in2 := #CI_UH31TA01ModeGoToRefPos)
      Contact( "STATUS_110".UH31_TA01.Specific.EposZSW2Detail.FixedStopReached )
      Move(in := #CI_UH31TA01ModeSetRefPos, out1 => #TS_UH31TA01.Mode)
   END_RUNG
   RUNG wire#powerrail
      Contact( "STATUS_110".UH31_TA01.Main.Man )
      Move(in := #CI_UH31TA01ModeJog, out1 => #TS_UH31TA01.Mode)
   END_RUNG
   // the same network as SCL:
   #TS_UH31TA01.Mode := #CI_UH31TA01ModeAbsPos;
   #_w1 := "JKU0Comm" AND "STATUS_Zone100".Station110_Mode.Main.Man;
   IF #_w1 AND "HMI_CMD_110".UH31_TA01_Ref THEN
       #TS_UH31TA01.Mode := #CI_UH31TA01ModeGoToRefPos;
       "HMI_CMD_110".UH31_TA01_Ref := FALSE;
   END_IF;
   IF #_w1 AND ("STATUS_110".UH31_TA01.Specific.ActMode = #CI_UH31TA01ModeGoToRefPos) AND "STATUS_110".UH31_TA01.Specific.EposZSW2Detail.FixedStopReached THEN
       #TS_UH31TA01.Mode := #CI_UH31TA01ModeSetRefPos;
   END_IF;
   IF "STATUS_110".UH31_TA01.Main.Man THEN #TS_UH31TA01.Mode := #CI_UH31TA01ModeJog; END_IF;
END_REGION

REGION Network 53: UH31-TA01 - FESTO servo - Parameters
   RUNG wire#powerrail
      { S7_Templates := "SrcType := Real" } Mul(in1 := #SR_UH31TA01SetPos, in2 := 1000.0, out => #TR_UH31TA01SetPos)
      { S7_Templates := "[SrcType := Real, DestType := DInt]" } Convert(in := #TR_UH31TA01SetPos, out => "HMI_PARAM_110".UH31_TA01.Position)
   END_RUNG
   RUNG wire#powerrail
      Move(in := 500, out1 => "HMI_PARAM_110".UH31_TA01.Velocity)
   END_RUNG
   RUNG wire#powerrail
      Move(in := 100, out1 => "HMI_PARAM_110".UH31_TA01.OverV)
      Move(in := 100, out1 => "HMI_PARAM_110".UH31_TA01.OverAcc)
      Move(in := 100, out1 => "HMI_PARAM_110".UH31_TA01.OverDec)
   END_RUNG
   // the same network as SCL:
   #TR_UH31TA01SetPos := #SR_UH31TA01SetPos * 1000.0;
   "HMI_PARAM_110".UH31_TA01.Position := REAL_TO_DINT(#TR_UH31TA01SetPos);
   "HMI_PARAM_110".UH31_TA01.Velocity := 500;
   "HMI_PARAM_110".UH31_TA01.OverV := 100;
   "HMI_PARAM_110".UH31_TA01.OverAcc := 100;
   "HMI_PARAM_110".UH31_TA01.OverDec := 100;
END_REGION

REGION Network 54: UH31-TA01 - STD_SERVO_FESTO_CMMT block call
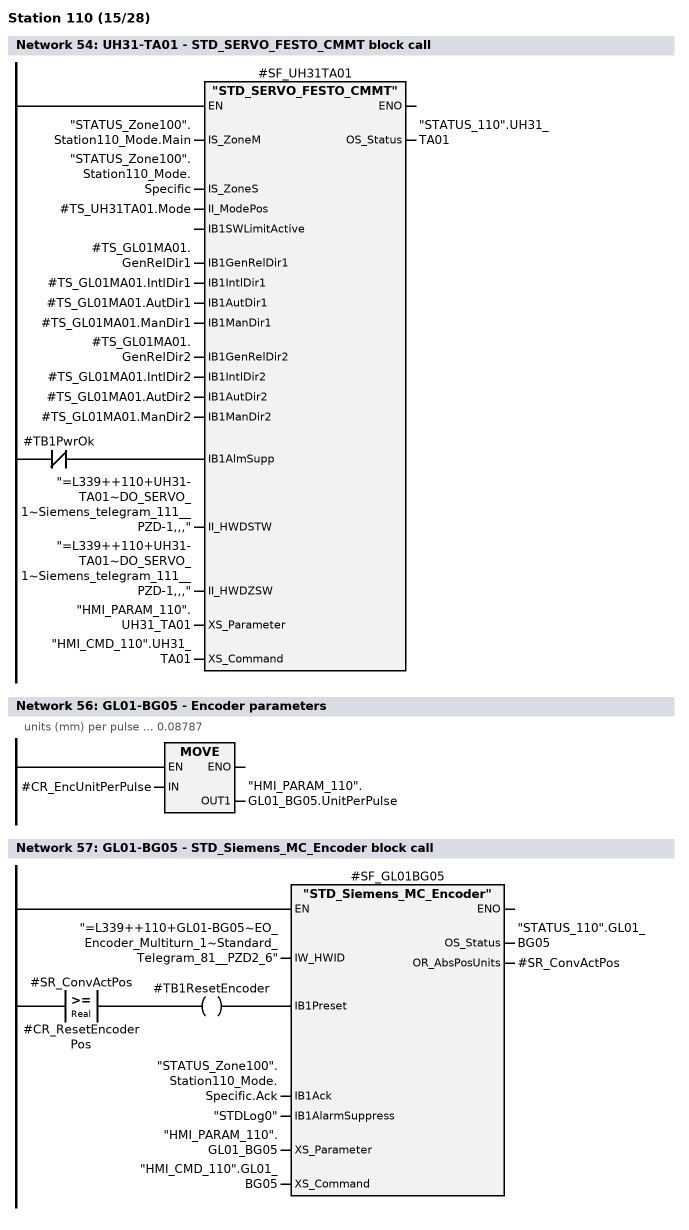
   RUNG wire#powerrail
      #SF_UH31TA01(IB1AlmSupp := wire#w1, IS_ZoneM := "STATUS_Zone100".Station110_Mode.Main, IS_ZoneS := "STATUS_Zone100".Station110_Mode.Specific, II_ModePos := #TS_UH31TA01.Mode, IB1SWLimitActive :=, IB1GenRelDir1 := #TS_GL01MA01.GenRelDir1, IB1IntlDir1 := #TS_GL01MA01.IntlDir1, IB1AutDir1 := #TS_GL01MA01.AutDir1, IB1ManDir1 := #TS_GL01MA01.ManDir1, IB1GenRelDir2 := #TS_GL01MA01.GenRelDir2, IB1IntlDir2 := #TS_GL01MA01.IntlDir2, IB1AutDir2 := #TS_GL01MA01.AutDir2, IB1ManDir2 := #TS_GL01MA01.ManDir2, II_HWDSTW := "=L339++110+UH31-TA01~DO_SERVO_1~Siemens_telegram_111__PZD-1,,,", II_HWDZSW := "=L339++110+UH31-TA01~DO_SERVO_1~Siemens_telegram_111__PZD-1,,,", XS_Parameter := "HMI_PARAM_110".UH31_TA01, XS_Command := "HMI_CMD_110".UH31_TA01, OS_Status => "STATUS_110".UH31_TA01)
   END_RUNG
   RUNG wire#powerrail
      I_Contact( #TB1PwrOk )
   END_RUNG wire#w1
   // the same network as SCL:
   #SF_UH31TA01(IS_ZoneM := "STATUS_Zone100".Station110_Mode.Main,   // "STD_SERVO_FESTO_CMMT"
                IS_ZoneS := "STATUS_Zone100".Station110_Mode.Specific,
                II_ModePos := #TS_UH31TA01.Mode,
                IB1GenRelDir1 := #TS_GL01MA01.GenRelDir1,
                IB1IntlDir1 := #TS_GL01MA01.IntlDir1,
                IB1AutDir1 := #TS_GL01MA01.AutDir1,
                IB1ManDir1 := #TS_GL01MA01.ManDir1,
                IB1GenRelDir2 := #TS_GL01MA01.GenRelDir2,
                IB1IntlDir2 := #TS_GL01MA01.IntlDir2,
                IB1AutDir2 := #TS_GL01MA01.AutDir2,
                IB1ManDir2 := #TS_GL01MA01.ManDir2,
                IB1AlmSupp := NOT #TB1PwrOk,
                II_HWDSTW := "=L339++110+UH31-TA01~DO_SERVO_1~Siemens_telegram_111__PZD-1,,,",
                II_HWDZSW := "=L339++110+UH31-TA01~DO_SERVO_1~Siemens_telegram_111__PZD-1,,,",
                XS_Parameter := "HMI_PARAM_110".UH31_TA01,
                XS_Command := "HMI_CMD_110".UH31_TA01,
                OS_Status => "STATUS_110".UH31_TA01);
END_REGION

REGION Network 55: *************** GL01-BG05 - Conveyor absolute encoder ***************
END_REGION

REGION Network 56: GL01-BG05 - Encoder parameters
   // units (mm) per pulse ... 0.08787
   RUNG wire#powerrail
      Move(in := #CR_EncUnitPerPulse, out1 => "HMI_PARAM_110".GL01_BG05.UnitPerPulse)
   END_RUNG
   // the same network as SCL:
   "HMI_PARAM_110".GL01_BG05.UnitPerPulse := #CR_EncUnitPerPulse;
END_REGION

REGION Network 57: GL01-BG05 - STD_Siemens_MC_Encoder block call
   RUNG wire#powerrail
      #SF_GL01BG05(IB1Preset := wire#w1, IW_HWID := "=L339++110+GL01-BG05~EO_Encoder_Multiturn_1~Standard_Telegram_81__PZD2_6", IB1Ack := "STATUS_Zone100".Station110_Mode.Specific.Ack, IB1AlarmSuppress := "STDLog0", XS_Parameter := "HMI_PARAM_110".GL01_BG05, XS_Command := "HMI_CMD_110".GL01_BG05, OS_Status => "STATUS_110".GL01_BG05, OR_AbsPosUnits => #SR_ConvActPos)
   END_RUNG
   RUNG wire#powerrail
      { S7_Templates := "SrcType := Real" } GE_Contact(in1 := #SR_ConvActPos, in2 := #CR_ResetEncoderPos)
      Coil( #TB1ResetEncoder )
   END_RUNG wire#w1
   // the same network as SCL:
   #TB1ResetEncoder := #SR_ConvActPos >= #CR_ResetEncoderPos;
   #SF_GL01BG05(IW_HWID := "=L339++110+GL01-BG05~EO_Encoder_Multiturn_1~Standard_Telegram_81__PZD2_6",   // "STD_Siemens_MC_Encoder"
                IB1Preset := #TB1ResetEncoder,
                IB1Ack := "STATUS_Zone100".Station110_Mode.Specific.Ack,
                IB1AlarmSuppress := "STDLog0",
                XS_Parameter := "HMI_PARAM_110".GL01_BG05,
                XS_Command := "HMI_CMD_110".GL01_BG05,
                OS_Status => "STATUS_110".GL01_BG05,
                OR_AbsPosUnits => #SR_ConvActPos);
END_REGION

REGION Network 58: *************** GL01-MA02 - Conveyor drive ***************
END_REGION

REGION Network 59: GL01-MA02 - Conveyor stop position
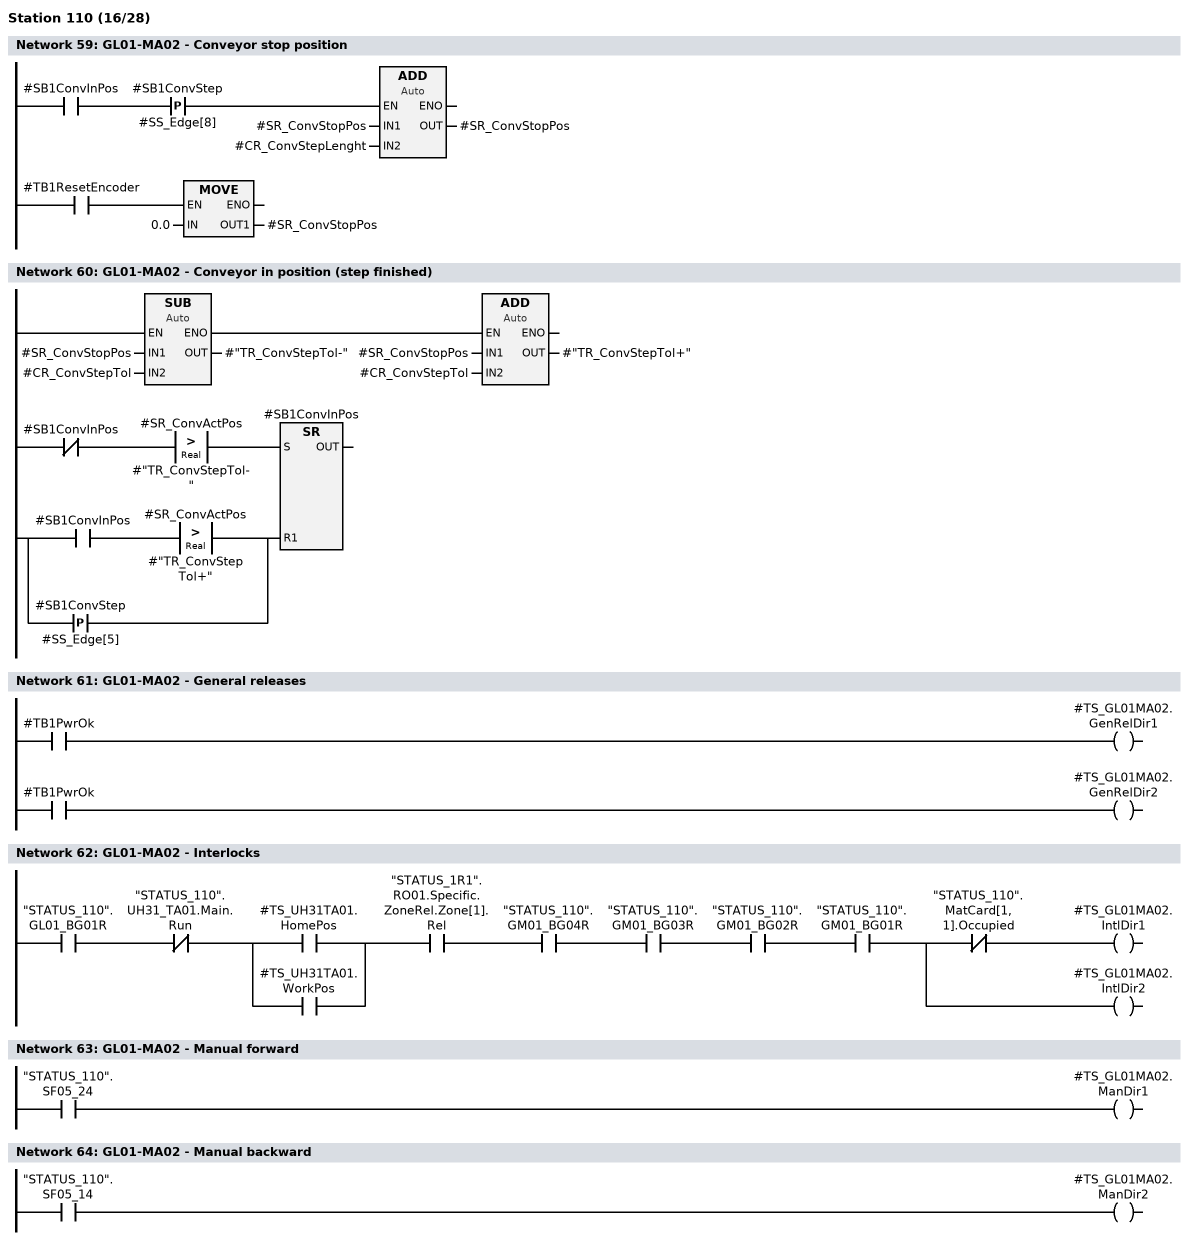
   RUNG wire#powerrail
      Contact( #SB1ConvInPos )
      P_Contact(operand := #SB1ConvStep, bit := #SS_Edge[8])
      Add(in1 := #SR_ConvStopPos, in2 := #CR_ConvStepLenght, out => #SR_ConvStopPos)
   END_RUNG
   RUNG wire#powerrail
      Contact( #TB1ResetEncoder )
      Move(in := 0.0, out1 => #SR_ConvStopPos)
   END_RUNG
   // the same network as SCL:
   #_w1 := #SB1ConvInPos AND #SB1ConvStep AND NOT #SS_Edge[8];   // rising edge of #SB1ConvStep
   #SS_Edge[8] := #SB1ConvStep;
   IF #_w1 THEN #SR_ConvStopPos := #SR_ConvStopPos + #CR_ConvStepLenght; END_IF;
   IF #TB1ResetEncoder THEN #SR_ConvStopPos := 0.0; END_IF;
END_REGION

REGION Network 60: GL01-MA02 - Conveyor in position (step finished)
   RUNG wire#powerrail
      Sub(in1 := #SR_ConvStopPos, in2 := #CR_ConvStepTol, out => #"TR_ConvStepTol-")
      Add(in1 := #SR_ConvStopPos, in2 := #CR_ConvStepTol, out => #"TR_ConvStepTol+")
   END_RUNG
   RUNG wire#powerrail
      I_Contact( #SB1ConvInPos )
      { S7_Templates := "SrcType := Real" } GT_Contact(in1 := #SR_ConvActPos, in2 := #"TR_ConvStepTol-")
      S_SR(operand := #SB1ConvInPos, r1 := wire#w1)
   END_RUNG
   RUNG wire#powerrail
      Contact( #SB1ConvInPos )
      { S7_Templates := "SrcType := Real" } GT_Contact(in1 := #SR_ConvActPos, in2 := #"TR_ConvStepTol+")
   END_RUNG wire#w1
   RUNG wire#powerrail
      P_Contact(operand := #SB1ConvStep, bit := #SS_Edge[5])
   END_RUNG wire#w1
   // the same network as SCL:
   #"TR_ConvStepTol-" := #SR_ConvStopPos - #CR_ConvStepTol;
   #"TR_ConvStepTol+" := #SR_ConvStopPos + #CR_ConvStepTol;
   #_w1 := #SB1ConvStep AND NOT #SS_Edge[5];   // rising edge of #SB1ConvStep
   #SS_Edge[5] := #SB1ConvStep;
   #_w2 := (#SB1ConvInPos AND (#SR_ConvActPos > #"TR_ConvStepTol+")) OR #_w1;
   IF NOT #SB1ConvInPos AND (#SR_ConvActPos > #"TR_ConvStepTol-") THEN
       #SB1ConvInPos := TRUE;   // SR flip-flop
   END_IF;
   IF #_w2 THEN #SB1ConvInPos := FALSE; END_IF;
END_REGION

REGION Network 61: GL01-MA02 - General releases
   RUNG wire#powerrail
      Contact( #TB1PwrOk )
      Coil( #TS_GL01MA02.GenRelDir1 )
   END_RUNG
   RUNG wire#powerrail
      Contact( #TB1PwrOk )
      Coil( #TS_GL01MA02.GenRelDir2 )
   END_RUNG
   // the same network as SCL:
   #TS_GL01MA02.GenRelDir1 := #TB1PwrOk;
   #TS_GL01MA02.GenRelDir2 := #TB1PwrOk;
END_REGION

REGION Network 62: GL01-MA02 - Interlocks
   RUNG wire#powerrail
      Contact( "STATUS_110".GL01_BG01R )
      I_Contact( "STATUS_110".UH31_TA01.Main.Run )
      wire#w1
      Contact( #TS_UH31TA01.HomePos )
      wire#w2
      Contact( "STATUS_1R1".RO01.Specific.ZoneRel.Zone[1].Rel )
      Contact( "STATUS_110".GM01_BG04R )
      Contact( "STATUS_110".GM01_BG03R )
      Contact( "STATUS_110".GM01_BG02R )
      Contact( "STATUS_110".GM01_BG01R )
      wire#w3
      I_Contact( "STATUS_110".MatCard[1, 1].Occupied )
      Coil( #TS_GL01MA02.IntlDir1 )
   END_RUNG
   RUNG wire#w1
      Contact( #TS_UH31TA01.WorkPos )
   END_RUNG wire#w2
   RUNG wire#w3
      Coil( #TS_GL01MA02.IntlDir2 )
   END_RUNG
   // the same network as SCL:
   #_w1 := "STATUS_110".GL01_BG01R AND NOT "STATUS_110".UH31_TA01.Main.Run AND (#TS_UH31TA01.HomePos OR #TS_UH31TA01.WorkPos) AND "STATUS_1R1".RO01.Specific.ZoneRel.Zone[1].Rel AND "STATUS_110".GM01_BG04R AND "STATUS_110".GM01_BG03R AND "STATUS_110".GM01_BG02R AND "STATUS_110".GM01_BG01R;
   #TS_GL01MA02.IntlDir1 := #_w1 AND NOT "STATUS_110".MatCard[1, 1].Occupied;
   #TS_GL01MA02.IntlDir2 := #_w1;
END_REGION

REGION Network 63: GL01-MA02 - Manual forward
   RUNG wire#powerrail
      Contact( "STATUS_110".SF05_24 )
      Coil( #TS_GL01MA02.ManDir1 )
   END_RUNG
   // the same network as SCL:
   #TS_GL01MA02.ManDir1 := "STATUS_110".SF05_24;
END_REGION

REGION Network 64: GL01-MA02 - Manual backward
   RUNG wire#powerrail
      Contact( "STATUS_110".SF05_14 )
      Coil( #TS_GL01MA02.ManDir2 )
   END_RUNG
   // the same network as SCL:
   #TS_GL01MA02.ManDir2 := "STATUS_110".SF05_14;
END_REGION

REGION Network 65: GL01-MA02 - Auto forward (stepping)
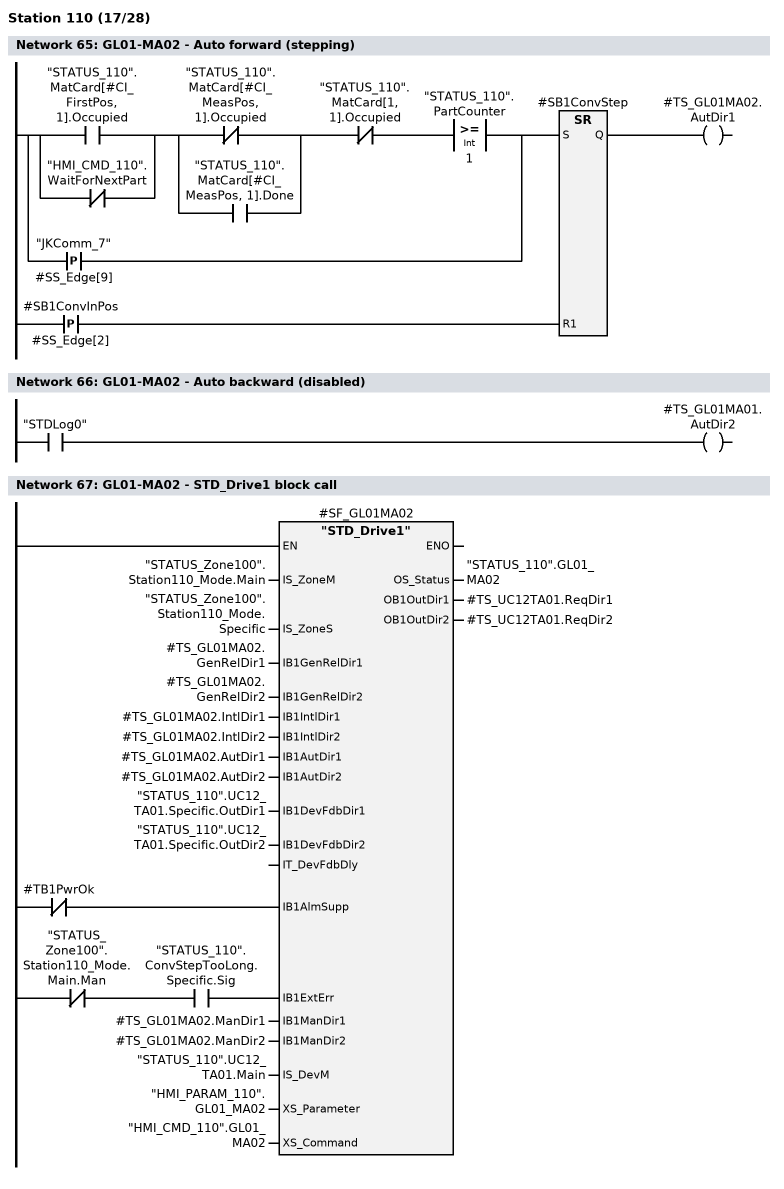
   RUNG wire#powerrail
      Contact( "STATUS_110".MatCard[#CI_FirstPos, 1].Occupied )
      wire#w1
      I_Contact( "STATUS_110".MatCard[#CI_MeasPos, 1].Occupied )
      wire#w2
      I_Contact( "STATUS_110".MatCard[1, 1].Occupied )
      { S7_Templates := "SrcType := Int" } GE_Contact(in1 := "STATUS_110".PartCounter, in2 := 1)
      wire#w3
      S_SR(operand := #SB1ConvStep, r1 := wire#w4)
      Coil( #TS_GL01MA02.AutDir1 )
   END_RUNG
   RUNG wire#powerrail
      I_Contact( "HMI_CMD_110".WaitForNextPart )
   END_RUNG wire#w1
   RUNG wire#w1
      Contact( "STATUS_110".MatCard[#CI_MeasPos, 1].Done )
   END_RUNG wire#w2
   RUNG wire#powerrail
      P_Contact(operand := "JKComm_7", bit := #SS_Edge[9])
   END_RUNG wire#w3
   RUNG wire#powerrail
      P_Contact(operand := #SB1ConvInPos, bit := #SS_Edge[2])
   END_RUNG wire#w4
   // the same network as SCL:
   #_w1 := "JKComm_7" AND NOT #SS_Edge[9];   // rising edge of "JKComm_7"
   #SS_Edge[9] := "JKComm_7";
   #_w2 := #SB1ConvInPos AND NOT #SS_Edge[2];   // rising edge of #SB1ConvInPos
   #SS_Edge[2] := #SB1ConvInPos;
   IF (("STATUS_110".MatCard[#CI_FirstPos, 1].Occupied OR NOT "HMI_CMD_110".WaitForNextPart) AND (NOT "STATUS_110".MatCard[#CI_MeasPos, 1].Occupied OR "STATUS_110".MatCard[#CI_MeasPos, 1].Done) AND NOT "STATUS_110".MatCard[1, 1].Occupied AND ("STATUS_110".PartCounter >= 1)) OR #_w1 THEN
       #SB1ConvStep := TRUE;   // SR flip-flop
   END_IF;
   IF #_w2 THEN #SB1ConvStep := FALSE; END_IF;
   #TS_GL01MA02.AutDir1 := #SB1ConvStep;
END_REGION

REGION Network 66: GL01-MA02 - Auto backward (disabled)
   RUNG wire#powerrail
      Contact( "STDLog0" )
      Coil( #TS_GL01MA01.AutDir2 )
   END_RUNG
   // the same network as SCL:
   #TS_GL01MA01.AutDir2 := "STDLog0";
END_REGION

REGION Network 67: GL01-MA02 - STD_Drive1 block call
   RUNG wire#powerrail
      #SF_GL01MA02(IB1AlmSupp := wire#w1, IB1ExtErr := wire#w2, IS_ZoneM := "STATUS_Zone100".Station110_Mode.Main, IS_ZoneS := "STATUS_Zone100".Station110_Mode.Specific, IB1GenRelDir1 := #TS_GL01MA02.GenRelDir1, IB1GenRelDir2 := #TS_GL01MA02.GenRelDir2, IB1IntlDir1 := #TS_GL01MA02.IntlDir1, IB1IntlDir2 := #TS_GL01MA02.IntlDir2, IB1AutDir1 := #TS_GL01MA02.AutDir1, IB1AutDir2 := #TS_GL01MA02.AutDir2, IB1DevFdbDir1 := "STATUS_110".UC12_TA01.Specific.OutDir1, IB1DevFdbDir2 := "STATUS_110".UC12_TA01.Specific.OutDir2, IT_DevFdbDly :=, IB1ManDir1 := #TS_GL01MA02.ManDir1, IB1ManDir2 := #TS_GL01MA02.ManDir2, IS_DevM := "STATUS_110".UC12_TA01.Main, XS_Parameter := "HMI_PARAM_110".GL01_MA02, XS_Command := "HMI_CMD_110".GL01_MA02, OS_Status => "STATUS_110".GL01_MA02, OB1OutDir1 => #TS_UC12TA01.ReqDir1, OB1OutDir2 => #TS_UC12TA01.ReqDir2)
   END_RUNG
   RUNG wire#powerrail
      I_Contact( #TB1PwrOk )
   END_RUNG wire#w1
   RUNG wire#powerrail
      I_Contact( "STATUS_Zone100".Station110_Mode.Main.Man )
      Contact( "STATUS_110".ConvStepTooLong.Specific.Sig )
   END_RUNG wire#w2
   // the same network as SCL:
   #SF_GL01MA02(IS_ZoneM := "STATUS_Zone100".Station110_Mode.Main,   // "STD_Drive1"
                IS_ZoneS := "STATUS_Zone100".Station110_Mode.Specific,
                IB1GenRelDir1 := #TS_GL01MA02.GenRelDir1,
                IB1GenRelDir2 := #TS_GL01MA02.GenRelDir2,
                IB1IntlDir1 := #TS_GL01MA02.IntlDir1,
                IB1IntlDir2 := #TS_GL01MA02.IntlDir2,
                IB1AutDir1 := #TS_GL01MA02.AutDir1,
                IB1AutDir2 := #TS_GL01MA02.AutDir2,
                IB1DevFdbDir1 := "STATUS_110".UC12_TA01.Specific.OutDir1,
                IB1DevFdbDir2 := "STATUS_110".UC12_TA01.Specific.OutDir2,
                IB1AlmSupp := NOT #TB1PwrOk,
                IB1ExtErr := NOT "STATUS_Zone100".Station110_Mode.Main.Man AND "STATUS_110".ConvStepTooLong.Specific.Sig,
                IB1ManDir1 := #TS_GL01MA02.ManDir1,
                IB1ManDir2 := #TS_GL01MA02.ManDir2,
                IS_DevM := "STATUS_110".UC12_TA01.Main,
                XS_Parameter := "HMI_PARAM_110".GL01_MA02,
                XS_Command := "HMI_CMD_110".GL01_MA02,
                OS_Status => "STATUS_110".GL01_MA02,
                OB1OutDir1 => #TS_UC12TA01.ReqDir1,
                OB1OutDir2 => #TS_UC12TA01.ReqDir2);
END_REGION

REGION Network 68: UC12-TA01 - Acknowledge error
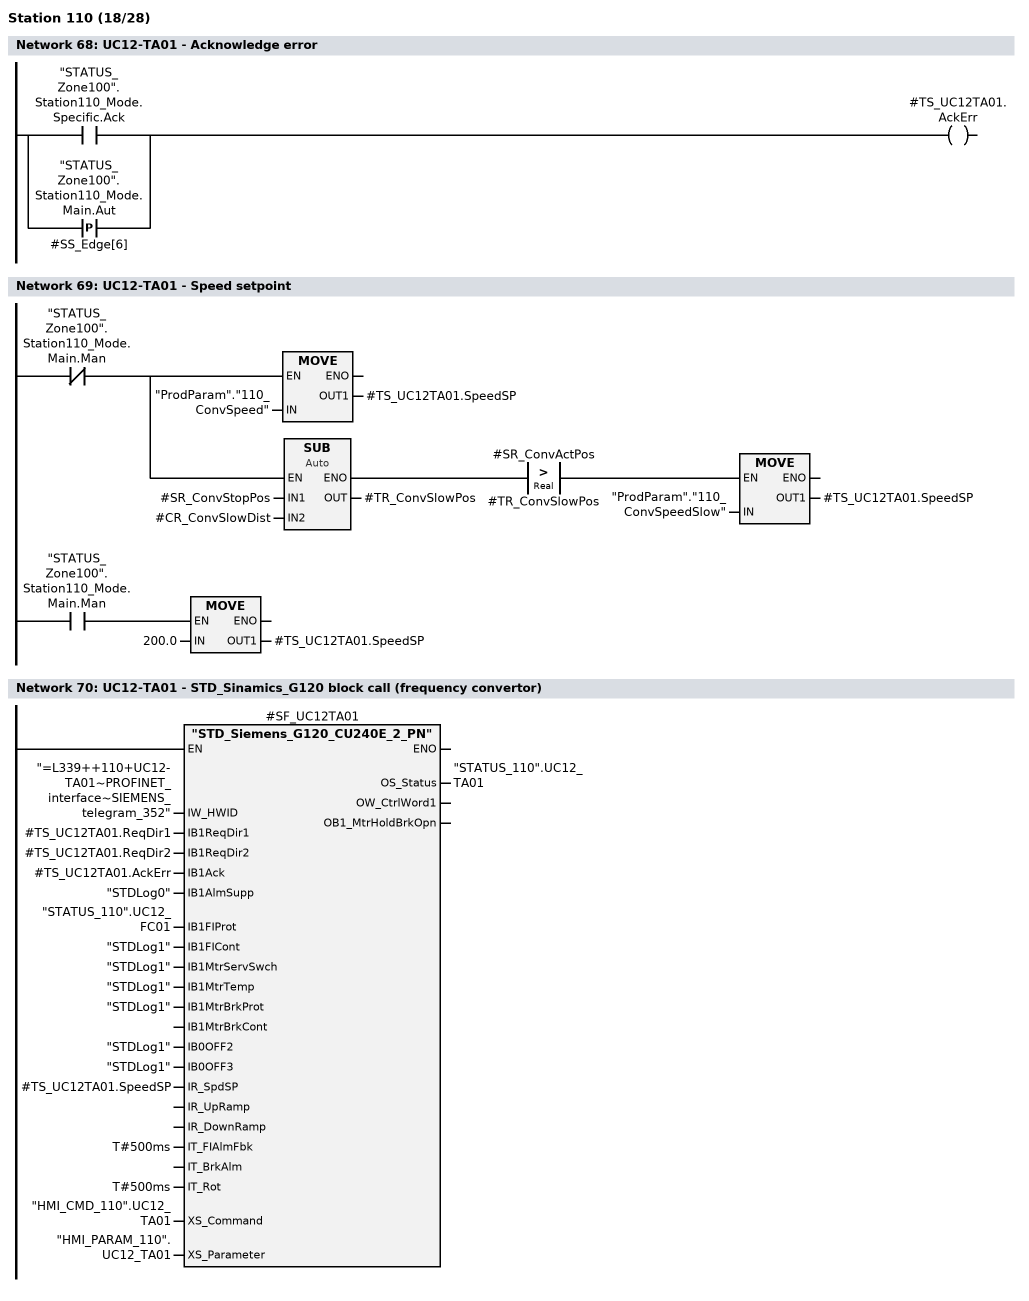
   RUNG wire#powerrail
      Contact( "STATUS_Zone100".Station110_Mode.Specific.Ack )
      wire#w1
      Coil( #TS_UC12TA01.AckErr )
   END_RUNG
   RUNG wire#powerrail
      P_Contact(operand := "STATUS_Zone100".Station110_Mode.Main.Aut, bit := #SS_Edge[6])
   END_RUNG wire#w1
   // the same network as SCL:
   #_w1 := "STATUS_Zone100".Station110_Mode.Main.Aut AND NOT #SS_Edge[6];   // rising edge of "STATUS_Zone100".Station110_Mode.Main.Aut
   #SS_Edge[6] := "STATUS_Zone100".Station110_Mode.Main.Aut;
   #TS_UC12TA01.AckErr := "STATUS_Zone100".Station110_Mode.Specific.Ack OR #_w1;
END_REGION

REGION Network 69: UC12-TA01 - Speed setpoint
   RUNG wire#powerrail
      I_Contact( "STATUS_Zone100".Station110_Mode.Main.Man )
      wire#w1
      Move(in := "ProdParam"."110_ConvSpeed", out1 => #TS_UC12TA01.SpeedSP)
   END_RUNG
   RUNG wire#w1
      Sub(in1 := #SR_ConvStopPos, in2 := #CR_ConvSlowDist, out => #TR_ConvSlowPos)
      { S7_Templates := "SrcType := Real" } GT_Contact(in1 := #SR_ConvActPos, in2 := #TR_ConvSlowPos)
      Move(in := "ProdParam"."110_ConvSpeedSlow", out1 => #TS_UC12TA01.SpeedSP)
   END_RUNG
   RUNG wire#powerrail
      Contact( "STATUS_Zone100".Station110_Mode.Main.Man )
      Move(in := 200.0, out1 => #TS_UC12TA01.SpeedSP)
   END_RUNG
   // the same network as SCL:
   #_w1 := NOT "STATUS_Zone100".Station110_Mode.Main.Man;
   IF #_w1 THEN
       #TS_UC12TA01.SpeedSP := "ProdParam"."110_ConvSpeed";
       #TR_ConvSlowPos := #SR_ConvStopPos - #CR_ConvSlowDist;
   END_IF;
   IF #_w1 AND (#SR_ConvActPos > #TR_ConvSlowPos) THEN
       #TS_UC12TA01.SpeedSP := "ProdParam"."110_ConvSpeedSlow";
   END_IF;
   IF "STATUS_Zone100".Station110_Mode.Main.Man THEN #TS_UC12TA01.SpeedSP := 200.0; END_IF;
END_REGION

REGION Network 70: UC12-TA01 - STD_Sinamics_G120 block call (frequency convertor)
   RUNG wire#powerrail
      #SF_UC12TA01(IW_HWID := "=L339++110+UC12-TA01~PROFINET_interface~SIEMENS_telegram_352", IB1ReqDir1 := #TS_UC12TA01.ReqDir1, IB1ReqDir2 := #TS_UC12TA01.ReqDir2, IB1Ack := #TS_UC12TA01.AckErr, IB1AlmSupp := "STDLog0", IB1FIProt := "STATUS_110".UC12_FC01, IB1FICont := "STDLog1", IB1MtrServSwch := "STDLog1", IB1MtrTemp := "STDLog1", IB1MtrBrkProt := "STDLog1", IB1MtrBrkCont :=, IB0OFF2 := "STDLog1", IB0OFF3 := "STDLog1", IR_SpdSP := #TS_UC12TA01.SpeedSP, IR_UpRamp :=, IR_DownRamp :=, IT_FIAlmFbk := T#500ms, IT_BrkAlm :=, IT_Rot := T#500ms, XS_Command := "HMI_CMD_110".UC12_TA01, XS_Parameter := "HMI_PARAM_110".UC12_TA01, OS_Status => "STATUS_110".UC12_TA01, OW_CtrlWord1 =>, OB1_MtrHoldBrkOpn =>)
   END_RUNG
   // the same network as SCL:
   #SF_UC12TA01(IW_HWID := "=L339++110+UC12-TA01~PROFINET_interface~SIEMENS_telegram_352",   // "STD_Siemens_G120_CU240E_2_PN"
                IB1ReqDir1 := #TS_UC12TA01.ReqDir1,
                IB1ReqDir2 := #TS_UC12TA01.ReqDir2,
                IB1Ack := #TS_UC12TA01.AckErr,
                IB1AlmSupp := "STDLog0",
                IB1FIProt := "STATUS_110".UC12_FC01,
                IB1FICont := "STDLog1",
                IB1MtrServSwch := "STDLog1",
                IB1MtrTemp := "STDLog1",
                IB1MtrBrkProt := "STDLog1",
                IB0OFF2 := "STDLog1",
                IB0OFF3 := "STDLog1",
                IR_SpdSP := #TS_UC12TA01.SpeedSP,
                IT_FIAlmFbk := T#500ms,
                IT_Rot := T#500ms,
                XS_Command := "HMI_CMD_110".UC12_TA01,
                XS_Parameter := "HMI_PARAM_110".UC12_TA01,
                OS_Status => "STATUS_110".UC12_TA01);
END_REGION

REGION Network 71: *************** GM01-MM04 - Lift 4 ***************
END_REGION

REGION Network 72: GM01-MM04 - General releases
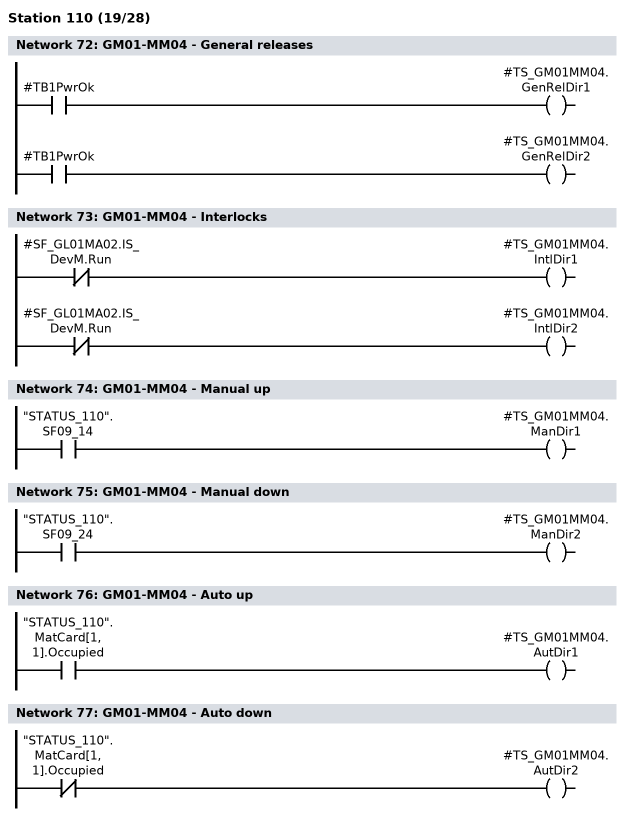
   RUNG wire#powerrail
      Contact( #TB1PwrOk )
      Coil( #TS_GM01MM04.GenRelDir1 )
   END_RUNG
   RUNG wire#powerrail
      Contact( #TB1PwrOk )
      Coil( #TS_GM01MM04.GenRelDir2 )
   END_RUNG
   // the same network as SCL:
   #TS_GM01MM04.GenRelDir1 := #TB1PwrOk;
   #TS_GM01MM04.GenRelDir2 := #TB1PwrOk;
END_REGION

REGION Network 73: GM01-MM04 - Interlocks
   RUNG wire#powerrail
      I_Contact( #SF_GL01MA02.IS_DevM.Run )
      Coil( #TS_GM01MM04.IntlDir1 )
   END_RUNG
   RUNG wire#powerrail
      I_Contact( #SF_GL01MA02.IS_DevM.Run )
      Coil( #TS_GM01MM04.IntlDir2 )
   END_RUNG
   // the same network as SCL:
   #TS_GM01MM04.IntlDir1 := NOT #SF_GL01MA02.IS_DevM.Run;
   #TS_GM01MM04.IntlDir2 := NOT #SF_GL01MA02.IS_DevM.Run;
END_REGION

REGION Network 74: GM01-MM04 - Manual up
   RUNG wire#powerrail
      Contact( "STATUS_110".SF09_14 )
      Coil( #TS_GM01MM04.ManDir1 )
   END_RUNG
   // the same network as SCL:
   #TS_GM01MM04.ManDir1 := "STATUS_110".SF09_14;
END_REGION

REGION Network 75: GM01-MM04 - Manual down
   RUNG wire#powerrail
      Contact( "STATUS_110".SF09_24 )
      Coil( #TS_GM01MM04.ManDir2 )
   END_RUNG
   // the same network as SCL:
   #TS_GM01MM04.ManDir2 := "STATUS_110".SF09_24;
END_REGION

REGION Network 76: GM01-MM04 - Auto up
   RUNG wire#powerrail
      Contact( "STATUS_110".MatCard[1, 1].Occupied )
      Coil( #TS_GM01MM04.AutDir1 )
   END_RUNG
   // the same network as SCL:
   #TS_GM01MM04.AutDir1 := "STATUS_110".MatCard[1, 1].Occupied;
END_REGION

REGION Network 77: GM01-MM04 - Auto down
   RUNG wire#powerrail
      I_Contact( "STATUS_110".MatCard[1, 1].Occupied )
      Coil( #TS_GM01MM04.AutDir2 )
   END_RUNG
   // the same network as SCL:
   #TS_GM01MM04.AutDir2 := NOT "STATUS_110".MatCard[1, 1].Occupied;
END_REGION

REGION Network 78: GM01-MM04 - Valve control
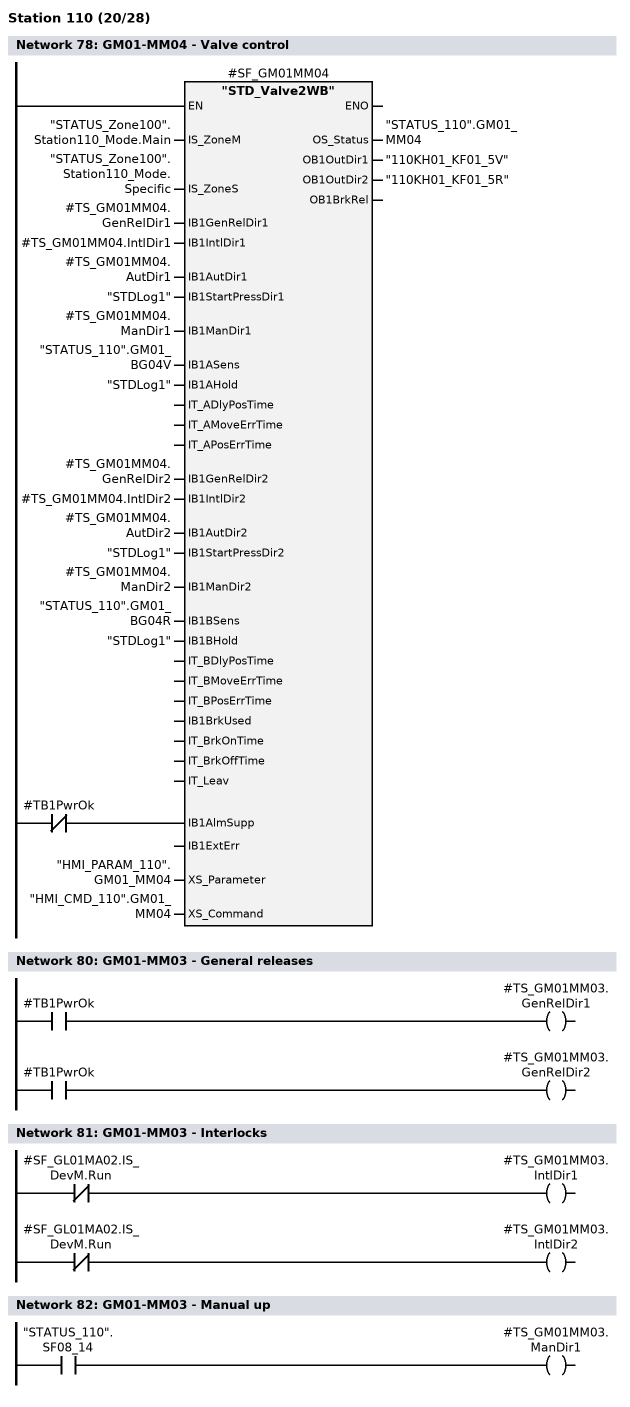
   RUNG wire#powerrail
      #SF_GM01MM04(IB1AlmSupp := wire#w1, IS_ZoneM := "STATUS_Zone100".Station110_Mode.Main, IS_ZoneS := "STATUS_Zone100".Station110_Mode.Specific, IB1GenRelDir1 := #TS_GM01MM04.GenRelDir1, IB1IntlDir1 := #TS_GM01MM04.IntlDir1, IB1AutDir1 := #TS_GM01MM04.AutDir1, IB1StartPressDir1 := "STDLog1", IB1ManDir1 := #TS_GM01MM04.ManDir1, IB1ASens := "STATUS_110".GM01_BG04V, IB1AHold := "STDLog1", IT_ADlyPosTime :=, IT_AMoveErrTime :=, IT_APosErrTime :=, IB1GenRelDir2 := #TS_GM01MM04.GenRelDir2, IB1IntlDir2 := #TS_GM01MM04.IntlDir2, IB1AutDir2 := #TS_GM01MM04.AutDir2, IB1StartPressDir2 := "STDLog1", IB1ManDir2 := #TS_GM01MM04.ManDir2, IB1BSens := "STATUS_110".GM01_BG04R, IB1BHold := "STDLog1", IT_BDlyPosTime :=, IT_BMoveErrTime :=, IT_BPosErrTime :=, IB1BrkUsed :=, IT_BrkOnTime :=, IT_BrkOffTime :=, IT_Leav :=, IB1ExtErr :=, XS_Parameter := "HMI_PARAM_110".GM01_MM04, XS_Command := "HMI_CMD_110".GM01_MM04, OS_Status => "STATUS_110".GM01_MM04, OB1OutDir1 => "110KH01_KF01_5V", OB1OutDir2 => "110KH01_KF01_5R", OB1BrkRel =>)
   END_RUNG
   RUNG wire#powerrail
      I_Contact( #TB1PwrOk )
   END_RUNG wire#w1
   // the same network as SCL:
   #SF_GM01MM04(IS_ZoneM := "STATUS_Zone100".Station110_Mode.Main,   // "STD_Valve2WB"
                IS_ZoneS := "STATUS_Zone100".Station110_Mode.Specific,
                IB1GenRelDir1 := #TS_GM01MM04.GenRelDir1,
                IB1IntlDir1 := #TS_GM01MM04.IntlDir1,
                IB1AutDir1 := #TS_GM01MM04.AutDir1,
                IB1StartPressDir1 := "STDLog1",
                IB1ManDir1 := #TS_GM01MM04.ManDir1,
                IB1ASens := "STATUS_110".GM01_BG04V,
                IB1AHold := "STDLog1",
                IB1GenRelDir2 := #TS_GM01MM04.GenRelDir2,
                IB1IntlDir2 := #TS_GM01MM04.IntlDir2,
                IB1AutDir2 := #TS_GM01MM04.AutDir2,
                IB1StartPressDir2 := "STDLog1",
                IB1ManDir2 := #TS_GM01MM04.ManDir2,
                IB1BSens := "STATUS_110".GM01_BG04R,
                IB1BHold := "STDLog1",
                IB1AlmSupp := NOT #TB1PwrOk,
                XS_Parameter := "HMI_PARAM_110".GM01_MM04,
                XS_Command := "HMI_CMD_110".GM01_MM04,
                OS_Status => "STATUS_110".GM01_MM04,
                OB1OutDir1 => "110KH01_KF01_5V",
                OB1OutDir2 => "110KH01_KF01_5R");
END_REGION

REGION Network 79: *************** GM01-MM03 - Lift 3 ***************
END_REGION

REGION Network 80: GM01-MM03 - General releases
   RUNG wire#powerrail
      Contact( #TB1PwrOk )
      Coil( #TS_GM01MM03.GenRelDir1 )
   END_RUNG
   RUNG wire#powerrail
      Contact( #TB1PwrOk )
      Coil( #TS_GM01MM03.GenRelDir2 )
   END_RUNG
   // the same network as SCL:
   #TS_GM01MM03.GenRelDir1 := #TB1PwrOk;
   #TS_GM01MM03.GenRelDir2 := #TB1PwrOk;
END_REGION

REGION Network 81: GM01-MM03 - Interlocks
   RUNG wire#powerrail
      I_Contact( #SF_GL01MA02.IS_DevM.Run )
      Coil( #TS_GM01MM03.IntlDir1 )
   END_RUNG
   RUNG wire#powerrail
      I_Contact( #SF_GL01MA02.IS_DevM.Run )
      Coil( #TS_GM01MM03.IntlDir2 )
   END_RUNG
   // the same network as SCL:
   #TS_GM01MM03.IntlDir1 := NOT #SF_GL01MA02.IS_DevM.Run;
   #TS_GM01MM03.IntlDir2 := NOT #SF_GL01MA02.IS_DevM.Run;
END_REGION

REGION Network 82: GM01-MM03 - Manual up
   RUNG wire#powerrail
      Contact( "STATUS_110".SF08_14 )
      Coil( #TS_GM01MM03.ManDir1 )
   END_RUNG
   // the same network as SCL:
   #TS_GM01MM03.ManDir1 := "STATUS_110".SF08_14;
END_REGION

REGION Network 83: GM01-MM03 - Manual down
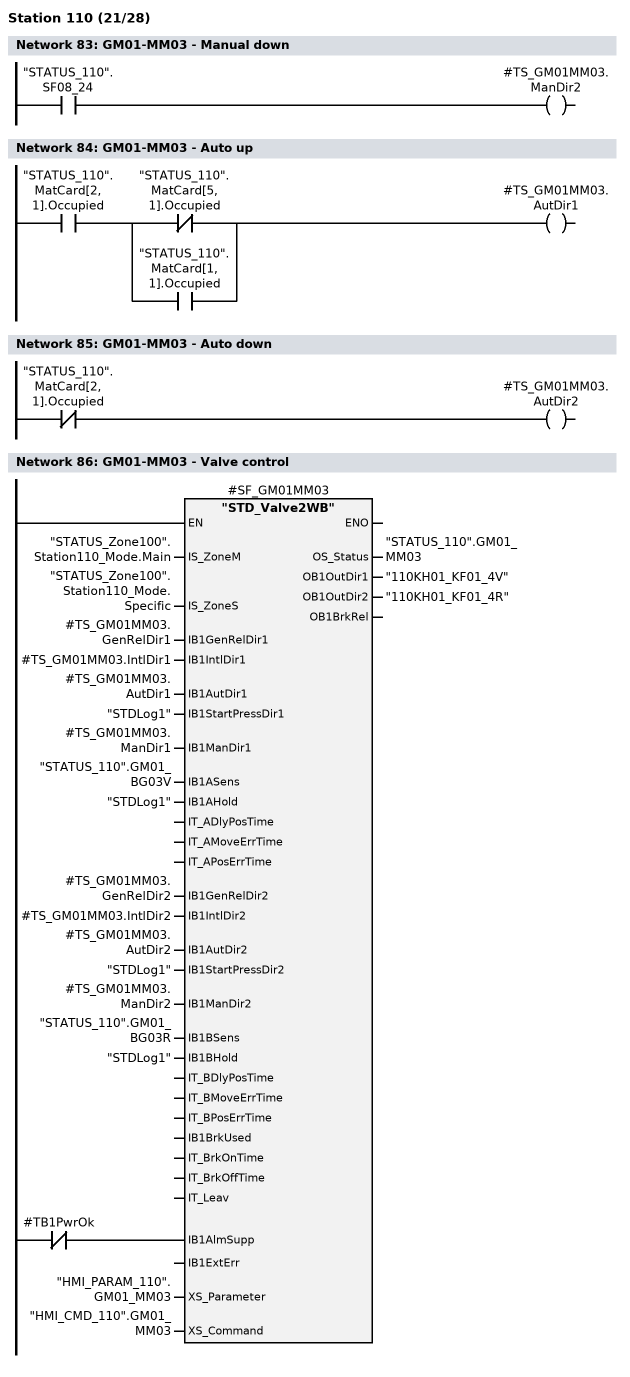
   RUNG wire#powerrail
      Contact( "STATUS_110".SF08_24 )
      Coil( #TS_GM01MM03.ManDir2 )
   END_RUNG
   // the same network as SCL:
   #TS_GM01MM03.ManDir2 := "STATUS_110".SF08_24;
END_REGION

REGION Network 84: GM01-MM03 - Auto up
   RUNG wire#powerrail
      Contact( "STATUS_110".MatCard[2, 1].Occupied )
      wire#w1
      I_Contact( "STATUS_110".MatCard[5, 1].Occupied )
      wire#w2
      Coil( #TS_GM01MM03.AutDir1 )
   END_RUNG
   RUNG wire#w1
      Contact( "STATUS_110".MatCard[1, 1].Occupied )
   END_RUNG wire#w2
   // the same network as SCL:
   #TS_GM01MM03.AutDir1 := "STATUS_110".MatCard[2, 1].Occupied AND (NOT "STATUS_110".MatCard[5, 1].Occupied OR "STATUS_110".MatCard[1, 1].Occupied);
END_REGION

REGION Network 85: GM01-MM03 - Auto down
   RUNG wire#powerrail
      I_Contact( "STATUS_110".MatCard[2, 1].Occupied )
      Coil( #TS_GM01MM03.AutDir2 )
   END_RUNG
   // the same network as SCL:
   #TS_GM01MM03.AutDir2 := NOT "STATUS_110".MatCard[2, 1].Occupied;
END_REGION

REGION Network 86: GM01-MM03 - Valve control
   RUNG wire#powerrail
      #SF_GM01MM03(IB1AlmSupp := wire#w1, IS_ZoneM := "STATUS_Zone100".Station110_Mode.Main, IS_ZoneS := "STATUS_Zone100".Station110_Mode.Specific, IB1GenRelDir1 := #TS_GM01MM03.GenRelDir1, IB1IntlDir1 := #TS_GM01MM03.IntlDir1, IB1AutDir1 := #TS_GM01MM03.AutDir1, IB1StartPressDir1 := "STDLog1", IB1ManDir1 := #TS_GM01MM03.ManDir1, IB1ASens := "STATUS_110".GM01_BG03V, IB1AHold := "STDLog1", IT_ADlyPosTime :=, IT_AMoveErrTime :=, IT_APosErrTime :=, IB1GenRelDir2 := #TS_GM01MM03.GenRelDir2, IB1IntlDir2 := #TS_GM01MM03.IntlDir2, IB1AutDir2 := #TS_GM01MM03.AutDir2, IB1StartPressDir2 := "STDLog1", IB1ManDir2 := #TS_GM01MM03.ManDir2, IB1BSens := "STATUS_110".GM01_BG03R, IB1BHold := "STDLog1", IT_BDlyPosTime :=, IT_BMoveErrTime :=, IT_BPosErrTime :=, IB1BrkUsed :=, IT_BrkOnTime :=, IT_BrkOffTime :=, IT_Leav :=, IB1ExtErr :=, XS_Parameter := "HMI_PARAM_110".GM01_MM03, XS_Command := "HMI_CMD_110".GM01_MM03, OS_Status => "STATUS_110".GM01_MM03, OB1OutDir1 => "110KH01_KF01_4V", OB1OutDir2 => "110KH01_KF01_4R", OB1BrkRel =>)
   END_RUNG
   RUNG wire#powerrail
      I_Contact( #TB1PwrOk )
   END_RUNG wire#w1
   // the same network as SCL:
   #SF_GM01MM03(IS_ZoneM := "STATUS_Zone100".Station110_Mode.Main,   // "STD_Valve2WB"
                IS_ZoneS := "STATUS_Zone100".Station110_Mode.Specific,
                IB1GenRelDir1 := #TS_GM01MM03.GenRelDir1,
                IB1IntlDir1 := #TS_GM01MM03.IntlDir1,
                IB1AutDir1 := #TS_GM01MM03.AutDir1,
                IB1StartPressDir1 := "STDLog1",
                IB1ManDir1 := #TS_GM01MM03.ManDir1,
                IB1ASens := "STATUS_110".GM01_BG03V,
                IB1AHold := "STDLog1",
                IB1GenRelDir2 := #TS_GM01MM03.GenRelDir2,
                IB1IntlDir2 := #TS_GM01MM03.IntlDir2,
                IB1AutDir2 := #TS_GM01MM03.AutDir2,
                IB1StartPressDir2 := "STDLog1",
                IB1ManDir2 := #TS_GM01MM03.ManDir2,
                IB1BSens := "STATUS_110".GM01_BG03R,
                IB1BHold := "STDLog1",
                IB1AlmSupp := NOT #TB1PwrOk,
                XS_Parameter := "HMI_PARAM_110".GM01_MM03,
                XS_Command := "HMI_CMD_110".GM01_MM03,
                OS_Status => "STATUS_110".GM01_MM03,
                OB1OutDir1 => "110KH01_KF01_4V",
                OB1OutDir2 => "110KH01_KF01_4R");
END_REGION

REGION Network 87: *************** GM01-MM02 - Lift 2 ***************
END_REGION

REGION Network 88: GM01-MM02 - General releases
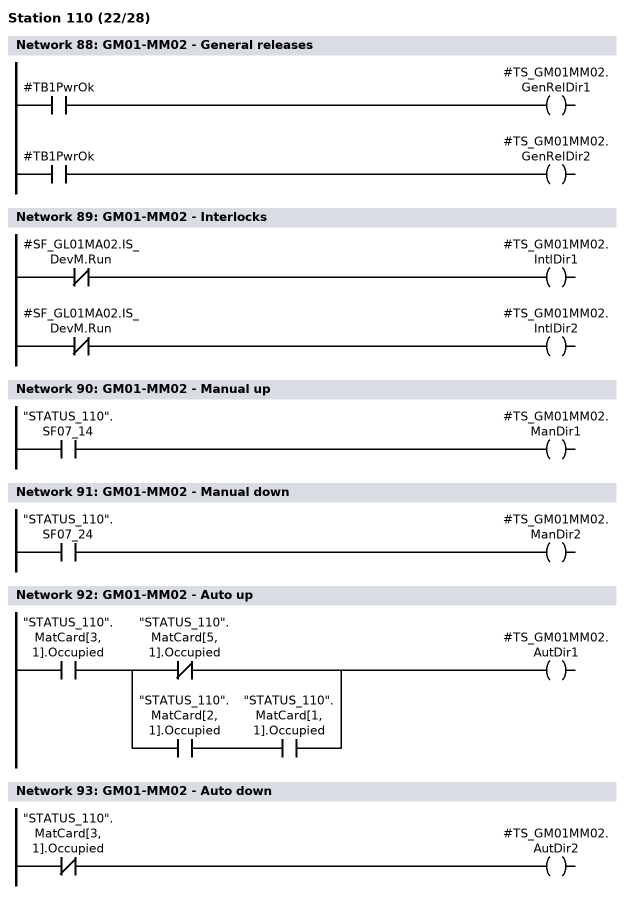
   RUNG wire#powerrail
      Contact( #TB1PwrOk )
      Coil( #TS_GM01MM02.GenRelDir1 )
   END_RUNG
   RUNG wire#powerrail
      Contact( #TB1PwrOk )
      Coil( #TS_GM01MM02.GenRelDir2 )
   END_RUNG
   // the same network as SCL:
   #TS_GM01MM02.GenRelDir1 := #TB1PwrOk;
   #TS_GM01MM02.GenRelDir2 := #TB1PwrOk;
END_REGION

REGION Network 89: GM01-MM02 - Interlocks
   RUNG wire#powerrail
      I_Contact( #SF_GL01MA02.IS_DevM.Run )
      Coil( #TS_GM01MM02.IntlDir1 )
   END_RUNG
   RUNG wire#powerrail
      I_Contact( #SF_GL01MA02.IS_DevM.Run )
      Coil( #TS_GM01MM02.IntlDir2 )
   END_RUNG
   // the same network as SCL:
   #TS_GM01MM02.IntlDir1 := NOT #SF_GL01MA02.IS_DevM.Run;
   #TS_GM01MM02.IntlDir2 := NOT #SF_GL01MA02.IS_DevM.Run;
END_REGION

REGION Network 90: GM01-MM02 - Manual up
   RUNG wire#powerrail
      Contact( "STATUS_110".SF07_14 )
      Coil( #TS_GM01MM02.ManDir1 )
   END_RUNG
   // the same network as SCL:
   #TS_GM01MM02.ManDir1 := "STATUS_110".SF07_14;
END_REGION

REGION Network 91: GM01-MM02 - Manual down
   RUNG wire#powerrail
      Contact( "STATUS_110".SF07_24 )
      Coil( #TS_GM01MM02.ManDir2 )
   END_RUNG
   // the same network as SCL:
   #TS_GM01MM02.ManDir2 := "STATUS_110".SF07_24;
END_REGION

REGION Network 92: GM01-MM02 - Auto up
   RUNG wire#powerrail
      Contact( "STATUS_110".MatCard[3, 1].Occupied )
      wire#w1
      I_Contact( "STATUS_110".MatCard[5, 1].Occupied )
      wire#w2
      Coil( #TS_GM01MM02.AutDir1 )
   END_RUNG
   RUNG wire#w1
      Contact( "STATUS_110".MatCard[2, 1].Occupied )
      Contact( "STATUS_110".MatCard[1, 1].Occupied )
   END_RUNG wire#w2
   // the same network as SCL:
   #TS_GM01MM02.AutDir1 := "STATUS_110".MatCard[3, 1].Occupied AND (NOT "STATUS_110".MatCard[5, 1].Occupied OR ("STATUS_110".MatCard[2, 1].Occupied AND "STATUS_110".MatCard[1, 1].Occupied));
END_REGION

REGION Network 93: GM01-MM02 - Auto down
   RUNG wire#powerrail
      I_Contact( "STATUS_110".MatCard[3, 1].Occupied )
      Coil( #TS_GM01MM02.AutDir2 )
   END_RUNG
   // the same network as SCL:
   #TS_GM01MM02.AutDir2 := NOT "STATUS_110".MatCard[3, 1].Occupied;
END_REGION

REGION Network 94: GM01-MM02 - Valve control
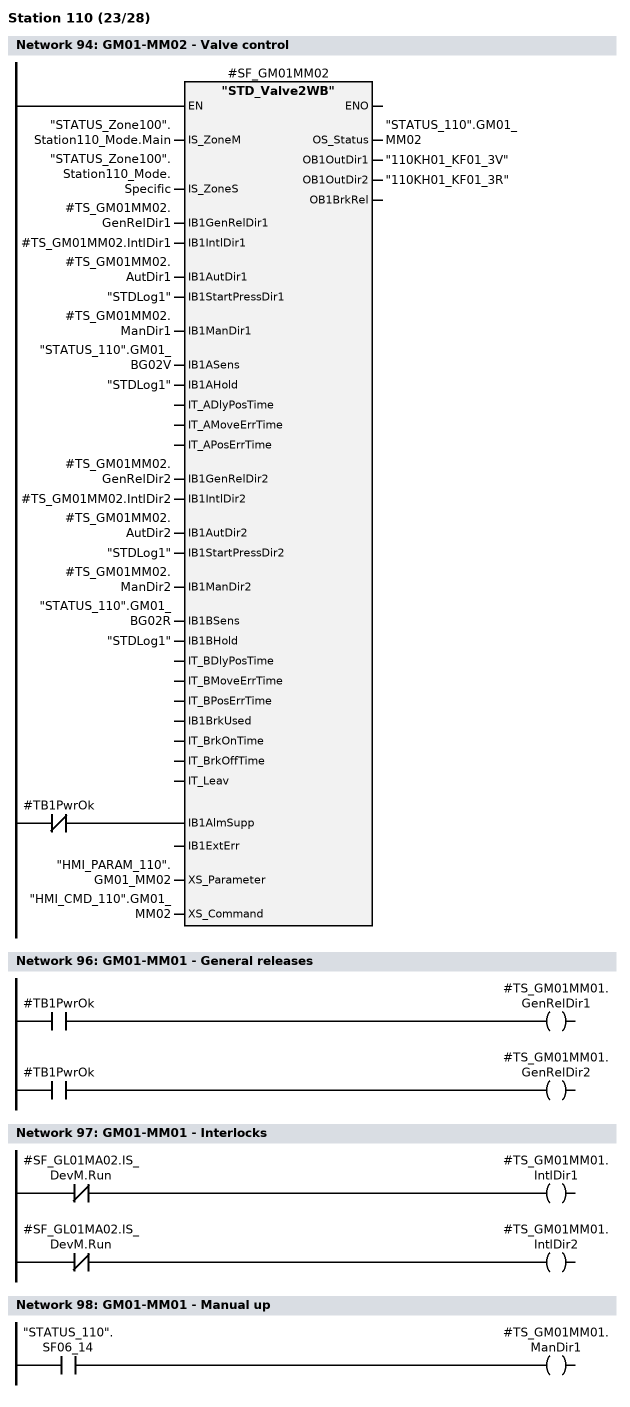
   RUNG wire#powerrail
      #SF_GM01MM02(IB1AlmSupp := wire#w1, IS_ZoneM := "STATUS_Zone100".Station110_Mode.Main, IS_ZoneS := "STATUS_Zone100".Station110_Mode.Specific, IB1GenRelDir1 := #TS_GM01MM02.GenRelDir1, IB1IntlDir1 := #TS_GM01MM02.IntlDir1, IB1AutDir1 := #TS_GM01MM02.AutDir1, IB1StartPressDir1 := "STDLog1", IB1ManDir1 := #TS_GM01MM02.ManDir1, IB1ASens := "STATUS_110".GM01_BG02V, IB1AHold := "STDLog1", IT_ADlyPosTime :=, IT_AMoveErrTime :=, IT_APosErrTime :=, IB1GenRelDir2 := #TS_GM01MM02.GenRelDir2, IB1IntlDir2 := #TS_GM01MM02.IntlDir2, IB1AutDir2 := #TS_GM01MM02.AutDir2, IB1StartPressDir2 := "STDLog1", IB1ManDir2 := #TS_GM01MM02.ManDir2, IB1BSens := "STATUS_110".GM01_BG02R, IB1BHold := "STDLog1", IT_BDlyPosTime :=, IT_BMoveErrTime :=, IT_BPosErrTime :=, IB1BrkUsed :=, IT_BrkOnTime :=, IT_BrkOffTime :=, IT_Leav :=, IB1ExtErr :=, XS_Parameter := "HMI_PARAM_110".GM01_MM02, XS_Command := "HMI_CMD_110".GM01_MM02, OS_Status => "STATUS_110".GM01_MM02, OB1OutDir1 => "110KH01_KF01_3V", OB1OutDir2 => "110KH01_KF01_3R", OB1BrkRel =>)
   END_RUNG
   RUNG wire#powerrail
      I_Contact( #TB1PwrOk )
   END_RUNG wire#w1
   // the same network as SCL:
   #SF_GM01MM02(IS_ZoneM := "STATUS_Zone100".Station110_Mode.Main,   // "STD_Valve2WB"
                IS_ZoneS := "STATUS_Zone100".Station110_Mode.Specific,
                IB1GenRelDir1 := #TS_GM01MM02.GenRelDir1,
                IB1IntlDir1 := #TS_GM01MM02.IntlDir1,
                IB1AutDir1 := #TS_GM01MM02.AutDir1,
                IB1StartPressDir1 := "STDLog1",
                IB1ManDir1 := #TS_GM01MM02.ManDir1,
                IB1ASens := "STATUS_110".GM01_BG02V,
                IB1AHold := "STDLog1",
                IB1GenRelDir2 := #TS_GM01MM02.GenRelDir2,
                IB1IntlDir2 := #TS_GM01MM02.IntlDir2,
                IB1AutDir2 := #TS_GM01MM02.AutDir2,
                IB1StartPressDir2 := "STDLog1",
                IB1ManDir2 := #TS_GM01MM02.ManDir2,
                IB1BSens := "STATUS_110".GM01_BG02R,
                IB1BHold := "STDLog1",
                IB1AlmSupp := NOT #TB1PwrOk,
                XS_Parameter := "HMI_PARAM_110".GM01_MM02,
                XS_Command := "HMI_CMD_110".GM01_MM02,
                OS_Status => "STATUS_110".GM01_MM02,
                OB1OutDir1 => "110KH01_KF01_3V",
                OB1OutDir2 => "110KH01_KF01_3R");
END_REGION

REGION Network 95: *************** GM01-MM01 - Lift 1 ***************
END_REGION

REGION Network 96: GM01-MM01 - General releases
   RUNG wire#powerrail
      Contact( #TB1PwrOk )
      Coil( #TS_GM01MM01.GenRelDir1 )
   END_RUNG
   RUNG wire#powerrail
      Contact( #TB1PwrOk )
      Coil( #TS_GM01MM01.GenRelDir2 )
   END_RUNG
   // the same network as SCL:
   #TS_GM01MM01.GenRelDir1 := #TB1PwrOk;
   #TS_GM01MM01.GenRelDir2 := #TB1PwrOk;
END_REGION

REGION Network 97: GM01-MM01 - Interlocks
   RUNG wire#powerrail
      I_Contact( #SF_GL01MA02.IS_DevM.Run )
      Coil( #TS_GM01MM01.IntlDir1 )
   END_RUNG
   RUNG wire#powerrail
      I_Contact( #SF_GL01MA02.IS_DevM.Run )
      Coil( #TS_GM01MM01.IntlDir2 )
   END_RUNG
   // the same network as SCL:
   #TS_GM01MM01.IntlDir1 := NOT #SF_GL01MA02.IS_DevM.Run;
   #TS_GM01MM01.IntlDir2 := NOT #SF_GL01MA02.IS_DevM.Run;
END_REGION

REGION Network 98: GM01-MM01 - Manual up
   RUNG wire#powerrail
      Contact( "STATUS_110".SF06_14 )
      Coil( #TS_GM01MM01.ManDir1 )
   END_RUNG
   // the same network as SCL:
   #TS_GM01MM01.ManDir1 := "STATUS_110".SF06_14;
END_REGION

REGION Network 99: GM01-MM01 - Manual down
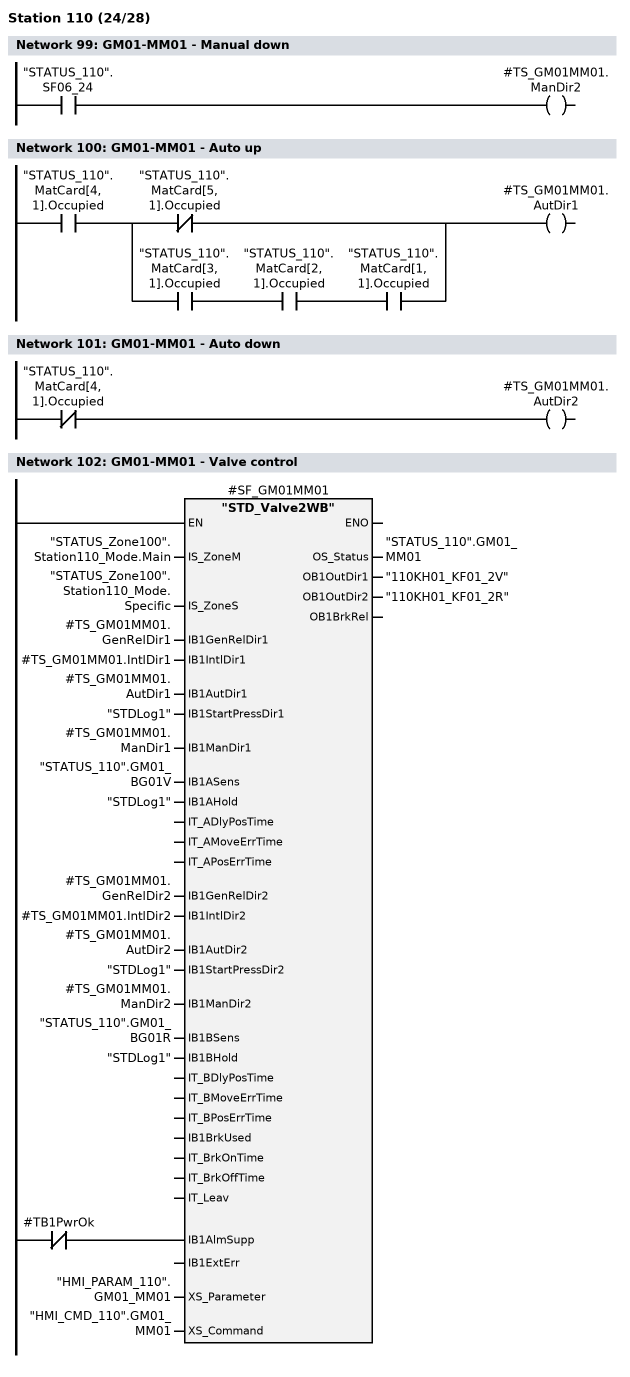
   RUNG wire#powerrail
      Contact( "STATUS_110".SF06_24 )
      Coil( #TS_GM01MM01.ManDir2 )
   END_RUNG
   // the same network as SCL:
   #TS_GM01MM01.ManDir2 := "STATUS_110".SF06_24;
END_REGION

REGION Network 100: GM01-MM01 - Auto up
   RUNG wire#powerrail
      Contact( "STATUS_110".MatCard[4, 1].Occupied )
      wire#w1
      I_Contact( "STATUS_110".MatCard[5, 1].Occupied )
      wire#w2
      Coil( #TS_GM01MM01.AutDir1 )
   END_RUNG
   RUNG wire#w1
      Contact( "STATUS_110".MatCard[3, 1].Occupied )
      Contact( "STATUS_110".MatCard[2, 1].Occupied )
      Contact( "STATUS_110".MatCard[1, 1].Occupied )
   END_RUNG wire#w2
   // the same network as SCL:
   #TS_GM01MM01.AutDir1 := "STATUS_110".MatCard[4, 1].Occupied AND (NOT "STATUS_110".MatCard[5, 1].Occupied OR ("STATUS_110".MatCard[3, 1].Occupied AND "STATUS_110".MatCard[2, 1].Occupied AND "STATUS_110".MatCard[1, 1].Occupied));
END_REGION

REGION Network 101: GM01-MM01 - Auto down
   RUNG wire#powerrail
      I_Contact( "STATUS_110".MatCard[4, 1].Occupied )
      Coil( #TS_GM01MM01.AutDir2 )
   END_RUNG
   // the same network as SCL:
   #TS_GM01MM01.AutDir2 := NOT "STATUS_110".MatCard[4, 1].Occupied;
END_REGION

REGION Network 102: GM01-MM01 - Valve control
   RUNG wire#powerrail
      #SF_GM01MM01(IB1AlmSupp := wire#w1, IS_ZoneM := "STATUS_Zone100".Station110_Mode.Main, IS_ZoneS := "STATUS_Zone100".Station110_Mode.Specific, IB1GenRelDir1 := #TS_GM01MM01.GenRelDir1, IB1IntlDir1 := #TS_GM01MM01.IntlDir1, IB1AutDir1 := #TS_GM01MM01.AutDir1, IB1StartPressDir1 := "STDLog1", IB1ManDir1 := #TS_GM01MM01.ManDir1, IB1ASens := "STATUS_110".GM01_BG01V, IB1AHold := "STDLog1", IT_ADlyPosTime :=, IT_AMoveErrTime :=, IT_APosErrTime :=, IB1GenRelDir2 := #TS_GM01MM01.GenRelDir2, IB1IntlDir2 := #TS_GM01MM01.IntlDir2, IB1AutDir2 := #TS_GM01MM01.AutDir2, IB1StartPressDir2 := "STDLog1", IB1ManDir2 := #TS_GM01MM01.ManDir2, IB1BSens := "STATUS_110".GM01_BG01R, IB1BHold := "STDLog1", IT_BDlyPosTime :=, IT_BMoveErrTime :=, IT_BPosErrTime :=, IB1BrkUsed :=, IT_BrkOnTime :=, IT_BrkOffTime :=, IT_Leav :=, IB1ExtErr :=, XS_Parameter := "HMI_PARAM_110".GM01_MM01, XS_Command := "HMI_CMD_110".GM01_MM01, OS_Status => "STATUS_110".GM01_MM01, OB1OutDir1 => "110KH01_KF01_2V", OB1OutDir2 => "110KH01_KF01_2R", OB1BrkRel =>)
   END_RUNG
   RUNG wire#powerrail
      I_Contact( #TB1PwrOk )
   END_RUNG wire#w1
   // the same network as SCL:
   #SF_GM01MM01(IS_ZoneM := "STATUS_Zone100".Station110_Mode.Main,   // "STD_Valve2WB"
                IS_ZoneS := "STATUS_Zone100".Station110_Mode.Specific,
                IB1GenRelDir1 := #TS_GM01MM01.GenRelDir1,
                IB1IntlDir1 := #TS_GM01MM01.IntlDir1,
                IB1AutDir1 := #TS_GM01MM01.AutDir1,
                IB1StartPressDir1 := "STDLog1",
                IB1ManDir1 := #TS_GM01MM01.ManDir1,
                IB1ASens := "STATUS_110".GM01_BG01V,
                IB1AHold := "STDLog1",
                IB1GenRelDir2 := #TS_GM01MM01.GenRelDir2,
                IB1IntlDir2 := #TS_GM01MM01.IntlDir2,
                IB1AutDir2 := #TS_GM01MM01.AutDir2,
                IB1StartPressDir2 := "STDLog1",
                IB1ManDir2 := #TS_GM01MM01.ManDir2,
                IB1BSens := "STATUS_110".GM01_BG01R,
                IB1BHold := "STDLog1",
                IB1AlmSupp := NOT #TB1PwrOk,
                XS_Parameter := "HMI_PARAM_110".GM01_MM01,
                XS_Command := "HMI_CMD_110".GM01_MM01,
                OS_Status => "STATUS_110".GM01_MM01,
                OB1OutDir1 => "110KH01_KF01_2V",
                OB1OutDir2 => "110KH01_KF01_2R");
END_REGION

REGION Network 103: *************** Material flow ***************
END_REGION

REGION Network 104: Part ID
